KUKA KRL program: f1_Kuka_APT209T03S09.SRC

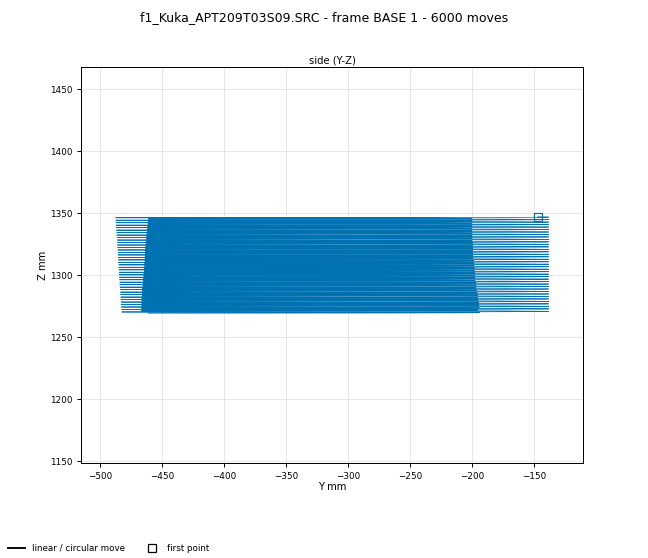
[picture p0: tool path of f1_Kuka_APT209T03S09.SRC in frame BASE 1, 6000 of 6001 moves have a stored position in this frame; points joined in program order, loops and branches not executed]
&ACCESS RVP
&REL 2
&PARAM TEMPLATE = C:\KRC\Roboter\Template\vorgabe
&PARAM EDITMASK = *
DEF f1_Kuka_APT209T03S09()


;FOLD INI;%{PE}%V3.2.0,%MKUKATPBASIS,%CINIT,%VCOMMON,%P
  ;FOLD BAS INI;%{E}%V3.2.0,%MKUKATPBASIS,%CINIT,%VINIT,%P
    GLOBAL INTERRUPT DECL 3 WHEN $STOPMESS==TRUE DO IR_STOPM ( )
    INTERRUPT ON 3
    BAS (#INITMOV,0 )
  ;ENDFOLD (BAS INI)
  ;FOLD USER INI;%{E}%V3.2.0,%MKUKATPUSER,%CINIT,%VINIT,%P
    ;Make your modifications here
  ;ENDFOLD (USER INI)
;ENDFOLD (INI)


;*** Make Null PTP Move
  PTP $pos_act

;*** Auto Load The Correct TOOL Data
  $tool=tool_data[3]

;*** Auto Load The Correct BASE Data
  $base=base_data[1]

  $ADVANCE = 5

;*** Restate Last Velocity
MMPM(30000.0)
SetRPM(6000)
LIN {X -0.021,Y -147.114,Z 1347.213,A 0.000,B 0.000,C 90.000,E1 218.382} C_DIS
LIN {X -0.029,Y -145.680,Z 1347.198,A 0.000,B 0.000,C 90.000,E1 215.644} C_DIS
LIN {X -0.031,Y -143.062,Z 1347.172,A 0.000,B 0.000,C 90.000,E1 211.052} C_DIS
LIN {X 0.026,Y -141.683,Z 1347.152,A 0.000,B 0.000,C 90.000,E1 207.334} C_DIS
LIN {X 0.005,Y -139.458,Z 1347.116,A 0.000,B 0.000,C 90.000,E1 200.844} C_DIS
LIN {X 0.056,Y -139.192,Z 1347.105,A 0.000,B 0.000,C 90.000,E1 198.960} C_DIS
LIN {X -0.057,Y -138.325,Z 1347.054,A 0.000,B 0.000,C 90.000,E1 189.670} C_DIS
LIN {X -0.053,Y -139.455,Z 1347.007,A 0.000,B 0.000,C 90.000,E1 181.260} C_DIS
LIN {X 0.027,Y -141.003,Z 1346.976,A 0.000,B 0.000,C 90.000,E1 175.641} C_DIS
LIN {X -0.023,Y -142.757,Z 1346.955,A 0.000,B 0.000,C 90.000,E1 171.951} C_DIS
LIN {X -0.068,Y -145.160,Z 1346.930,A 0.000,B 0.000,C 90.000,E1 167.353} C_DIS
LIN {X -0.076,Y -147.782,Z 1346.909,A 0.000,B 0.000,C 90.000,E1 163.685} C_DIS
LIN {X 0.003,Y -150.461,Z 1346.889,A 0.000,B 0.000,C 90.000,E1 160.007} C_DIS
LIN {X 0.079,Y -153.912,Z 1346.869,A 0.000,B 0.000,C 90.000,E1 156.357} C_DIS
LIN {X 0.003,Y -157.323,Z 1346.849,A 0.000,B 0.000,C 90.000,E1 152.794} C_DIS
LIN {X 0.087,Y -161.511,Z 1346.829,A 0.000,B 0.000,C 90.000,E1 149.203} C_DIS
LIN {X -0.036,Y -165.710,Z 1346.809,A 0.000,B 0.000,C 90.000,E1 145.722} C_DIS
LIN {X 0.089,Y -170.656,Z 1346.790,A 0.000,B 0.000,C 90.000,E1 142.190} C_DIS
LIN {X 0.002,Y -175.533,Z 1346.771,A 0.000,B 0.000,C 90.000,E1 138.771} C_DIS
LIN {X -0.004,Y -181.152,Z 1346.752,A 0.000,B 0.000,C 90.000,E1 135.364} C_DIS
LIN {X -0.007,Y -186.605,Z 1346.733,A 0.000,B 0.000,C 90.000,E1 132.000} C_DIS
LIN {X 0.063,Y -191.214,Z 1346.719,A 0.000,B 0.000,C 90.000,E1 129.483} C_DIS
LIN {X -0.013,Y -197.028,Z 1346.701,A 0.000,B 0.000,C 90.000,E1 126.217} C_DIS
LIN {X 0.060,Y -199.188,Z 1346.695,A 0.000,B 0.000,C 90.000,E1 125.105} C_DIS
LIN {X 0.058,Y -308.836,Z 1346.695,A 0.000,B 0.000,C 90.000,E1 125.105} C_DIS
LIN {X -0.131,Y -311.015,Z 1346.695,A 0.000,B 0.000,C 90.000,E1 125.105} C_DIS
LIN {X 0.079,Y -315.979,Z 1346.693,A 0.000,B 0.000,C 90.000,E1 124.818} C_DIS
LIN {X -0.152,Y -318.679,Z 1346.692,A 0.000,B 0.000,C 90.000,E1 124.612} C_DIS
LIN {X -0.061,Y -322.397,Z 1346.689,A 0.000,B 0.000,C 90.000,E1 124.072} C_DIS
LIN {X 0.196,Y -323.974,Z 1346.688,A 0.000,B 0.000,C 90.000,E1 123.706} C_DIS
LIN {X 0.124,Y -329.656,Z 1346.679,A 0.000,B 0.000,C 90.000,E1 122.133} C_DIS
LIN {X 0.058,Y -340.607,Z 1346.663,A 0.000,B 0.000,C 90.000,E1 119.333} C_DIS
LIN {X 0.113,Y -352.941,Z 1346.648,A 0.000,B 0.000,C 90.000,E1 116.565} C_DIS
LIN {X -0.104,Y -366.760,Z 1346.633,A 0.000,B 0.000,C 90.000,E1 113.898} C_DIS
LIN {X -0.018,Y -380.391,Z 1346.620,A 0.000,B 0.000,C 90.000,E1 111.535} C_DIS
LIN {X 0.139,Y -395.388,Z 1346.607,A 0.000,B 0.000,C 90.000,E1 109.214} C_DIS
LIN {X 0.038,Y -411.854,Z 1346.594,A 0.000,B 0.000,C 90.000,E1 106.985} C_DIS
LIN {X 0.222,Y -429.907,Z 1346.582,A 0.000,B 0.000,C 90.000,E1 104.773} C_DIS
LIN {X -0.080,Y -449.484,Z 1346.571,A 0.000,B 0.000,C 90.000,E1 102.703} C_DIS
LIN {X 0.151,Y -469.762,Z 1346.560,A 0.000,B 0.000,C 90.000,E1 100.725} C_DIS
LIN {X -0.162,Y -480.082,Z 1346.555,A 0.000,B 0.000,C 90.000,E1 99.849} C_DIS
LIN {X -0.063,Y -482.184,Z 1346.553,A 0.000,B 0.000,C 90.000,E1 99.613} C_DIS
LIN {X -0.184,Y -483.945,Z 1346.552,A 0.000,B 0.000,C 90.000,E1 99.378} C_DIS
LIN {X 0.095,Y -485.266,Z 1346.551,A 0.000,B 0.000,C 90.000,E1 99.095} C_DIS
LIN {X -0.127,Y -486.906,Z 1346.548,A 0.000,B 0.000,C 90.000,E1 98.624} C_DIS
LIN {X 0.065,Y -487.471,Z 1346.545,A 0.000,B 0.000,C 90.000,E1 98.106} C_DIS
LIN {X -0.214,Y -487.053,Z 1346.542,A 0.000,B 0.000,C 90.000,E1 97.644} C_DIS
LIN {X -0.007,Y -485.591,Z 1346.540,A 0.000,B 0.000,C 90.000,E1 97.125} C_DIS
LIN {X -0.116,Y -484.390,Z 1346.538,A 0.000,B 0.000,C 90.000,E1 96.891} C_DIS
LIN {X 0.079,Y -480.928,Z 1346.535,A 0.000,B 0.000,C 90.000,E1 96.372} C_DIS
LIN {X -0.128,Y -468.644,Z 1346.526,A 0.000,B 0.000,C 90.000,E1 94.645} C_DIS
LIN {X -0.194,Y -460.372,Z 1346.519,A 0.000,B 0.000,C 90.000,E1 93.383} C_DIS
LIN {X -0.018,Y -442.160,Z 1346.503,A 0.000,B 0.000,C 90.000,E1 90.516} C_DIS
LIN {X -0.118,Y -427.307,Z 1346.488,A 0.000,B 0.000,C 90.000,E1 87.879} C_DIS
LIN {X -0.104,Y -417.153,Z 1346.478,A 0.000,B 0.000,C 90.000,E1 85.988} C_DIS
LIN {X 0.161,Y -406.849,Z 1346.467,A 0.000,B 0.000,C 90.000,E1 84.033} C_DIS
LIN {X -0.175,Y -397.806,Z 1346.458,A 0.000,B 0.000,C 90.000,E1 82.413} C_DIS
LIN {X 0.118,Y -388.604,Z 1346.448,A 0.000,B 0.000,C 90.000,E1 80.679} C_DIS
LIN {X -0.083,Y -379.155,Z 1346.439,A 0.000,B 0.000,C 90.000,E1 78.993} C_DIS
LIN {X 0.068,Y -369.496,Z 1346.429,A 0.000,B 0.000,C 90.000,E1 77.229} C_DIS
LIN {X 0.006,Y -357.966,Z 1346.418,A 0.000,B 0.000,C 90.000,E1 75.172} C_DIS
LIN {X -0.113,Y -346.459,Z 1346.406,A 0.000,B 0.000,C 90.000,E1 73.087} C_DIS
LIN {X 0.053,Y -334.769,Z 1346.394,A 0.000,B 0.000,C 90.000,E1 70.913} C_DIS
LIN {X 0.078,Y -323.286,Z 1346.382,A 0.000,B 0.000,C 90.000,E1 68.720} C_DIS
LIN {X -0.120,Y -306.185,Z 1346.362,A 0.000,B 0.000,C 90.000,E1 65.229} C_DIS
LIN {X -0.076,Y -296.339,Z 1346.349,A 0.000,B 0.000,C 90.000,E1 62.922} C_DIS
LIN {X -0.095,Y -288.786,Z 1346.338,A 0.000,B 0.000,C 90.000,E1 60.923} C_DIS
LIN {X 0.023,Y -281.931,Z 1346.327,A 0.000,B 0.000,C 90.000,E1 58.869} C_DIS
LIN {X -0.138,Y -271.800,Z 1346.308,A 0.000,B 0.000,C 90.000,E1 55.468} C_DIS
LIN {X -0.041,Y -262.409,Z 1346.289,A 0.000,B 0.000,C 90.000,E1 51.949} C_DIS
LIN {X -0.118,Y -253.519,Z 1346.269,A 0.000,B 0.000,C 90.000,E1 48.405} C_DIS
LIN {X -0.011,Y -245.175,Z 1346.249,A 0.000,B 0.000,C 90.000,E1 44.757} C_DIS
LIN {X 0.013,Y -237.527,Z 1346.228,A 0.000,B 0.000,C 90.000,E1 41.067} C_DIS
LIN {X 0.054,Y -230.665,Z 1346.207,A 0.000,B 0.000,C 90.000,E1 37.317} C_DIS
LIN {X 0.153,Y -224.658,Z 1346.186,A 0.000,B 0.000,C 90.000,E1 33.499} C_DIS
LIN {X 0.131,Y -219.690,Z 1346.165,A 0.000,B 0.000,C 90.000,E1 29.667} C_DIS
LIN {X 0.066,Y -215.042,Z 1346.139,A 0.000,B 0.000,C 90.000,E1 25.027} C_DIS
LIN {X -0.033,Y -211.493,Z 1346.113,A 0.000,B 0.000,C 90.000,E1 20.355} C_DIS
LIN {X 0.064,Y -208.962,Z 1346.091,A 0.000,B 0.000,C 90.000,E1 16.386} C_DIS
LIN {X 0.106,Y -206.550,Z 1346.069,A 0.000,B 0.000,C 90.000,E1 12.411} C_DIS
LIN {X 0.007,Y -204.341,Z 1346.047,A 0.000,B 0.000,C 90.000,E1 8.454} C_DIS
LIN {X -0.064,Y -202.124,Z 1346.020,A 0.000,B 0.000,C 90.000,E1 3.669} C_DIS
LIN {X -0.057,Y -200.683,Z 1345.988,A 0.000,B 0.000,C 90.000,E1 357.936} C_DIS
LIN {X -0.077,Y -200.557,Z 1345.953,A 0.000,B 0.000,C 90.000,E1 351.489} C_DIS
LIN {X 0.019,Y -202.765,Z 1345.912,A 0.000,B 0.000,C 90.000,E1 344.212} C_DIS
LIN {X 0.067,Y -206.427,Z 1345.881,A 0.000,B 0.000,C 90.000,E1 338.592} C_DIS
LIN {X -0.106,Y -210.232,Z 1345.859,A 0.000,B 0.000,C 90.000,E1 334.665} C_DIS
LIN {X -0.083,Y -215.076,Z 1345.837,A 0.000,B 0.000,C 90.000,E1 330.717} C_DIS
LIN {X 0.041,Y -221.062,Z 1345.816,A 0.000,B 0.000,C 90.000,E1 326.786} C_DIS
LIN {X 0.102,Y -228.174,Z 1345.794,A 0.000,B 0.000,C 90.000,E1 322.924} C_DIS
LIN {X -0.060,Y -236.414,Z 1345.773,A 0.000,B 0.000,C 90.000,E1 319.175} C_DIS
LIN {X -0.018,Y -244.846,Z 1345.755,A 0.000,B 0.000,C 90.000,E1 315.810} C_DIS
LIN {X 0.115,Y -253.283,Z 1345.738,A 0.000,B 0.000,C 90.000,E1 312.852} C_DIS
LIN {X -0.047,Y -263.012,Z 1345.722,A 0.000,B 0.000,C 90.000,E1 310.011} C_DIS
LIN {X 0.023,Y -272.626,Z 1345.708,A 0.000,B 0.000,C 90.000,E1 307.523} C_DIS
LIN {X -0.011,Y -283.429,Z 1345.695,A 0.000,B 0.000,C 90.000,E1 305.105} C_DIS
LIN {X 0.139,Y -291.935,Z 1345.686,A 0.000,B 0.000,C 90.000,E1 303.372} C_DIS
LIN {X 0.030,Y -303.488,Z 1345.674,A 0.000,B 0.000,C 90.000,E1 301.386} C_DIS
LIN {X -0.014,Y -312.061,Z 1345.667,A 0.000,B 0.000,C 90.000,E1 300.079} C_DIS
LIN {X 0.060,Y -321.507,Z 1345.660,A 0.000,B 0.000,C 90.000,E1 298.771} C_DIS
LIN {X -0.126,Y -339.453,Z 1345.648,A 0.000,B 0.000,C 90.000,E1 296.616} C_DIS
LIN {X 0.065,Y -355.465,Z 1345.638,A 0.000,B 0.000,C 90.000,E1 294.771} C_DIS
LIN {X -0.108,Y -368.559,Z 1345.630,A 0.000,B 0.000,C 90.000,E1 293.334} C_DIS
LIN {X 0.060,Y -378.763,Z 1345.623,A 0.000,B 0.000,C 90.000,E1 292.153} C_DIS
LIN {X -0.141,Y -391.154,Z 1345.615,A 0.000,B 0.000,C 90.000,E1 290.737} C_DIS
LIN {X 0.096,Y -408.316,Z 1345.604,A 0.000,B 0.000,C 90.000,E1 288.725} C_DIS
LIN {X 0.076,Y -420.515,Z 1345.596,A 0.000,B 0.000,C 90.000,E1 287.347} C_DIS
LIN {X 0.078,Y -429.793,Z 1345.590,A 0.000,B 0.000,C 90.000,E1 286.260} C_DIS
LIN {X -0.126,Y -436.230,Z 1345.586,A 0.000,B 0.000,C 90.000,E1 285.481} C_DIS
LIN {X 0.040,Y -442.070,Z 1345.582,A 0.000,B 0.000,C 90.000,E1 284.662} C_DIS
LIN {X -0.060,Y -447.229,Z 1345.577,A 0.000,B 0.000,C 90.000,E1 283.883} C_DIS
LIN {X 0.216,Y -451.529,Z 1345.573,A 0.000,B 0.000,C 90.000,E1 283.063} C_DIS
LIN {X 0.091,Y -455.098,Z 1345.568,A 0.000,B 0.000,C 90.000,E1 282.299} C_DIS
LIN {X 0.175,Y -457.056,Z 1345.566,A 0.000,B 0.000,C 90.000,E1 281.771} C_DIS
LIN {X -0.185,Y -458.644,Z 1345.563,A 0.000,B 0.000,C 90.000,E1 281.299} C_DIS
LIN {X -0.174,Y -459.895,Z 1345.560,A 0.000,B 0.000,C 90.000,E1 280.782} C_DIS
LIN {X -0.064,Y -460.730,Z 1345.557,A 0.000,B 0.000,C 90.000,E1 280.254} C_DIS
LIN {X 0.049,Y -461.072,Z 1345.554,A 0.000,B 0.000,C 90.000,E1 279.726} C_DIS
LIN {X 0.090,Y -460.985,Z 1345.551,A 0.000,B 0.000,C 90.000,E1 279.208} C_DIS
LIN {X 0.136,Y -460.415,Z 1345.548,A 0.000,B 0.000,C 90.000,E1 278.690} C_DIS
LIN {X -0.204,Y -459.357,Z 1345.546,A 0.000,B 0.000,C 90.000,E1 278.219} C_DIS
LIN {X -0.161,Y -457.815,Z 1345.543,A 0.000,B 0.000,C 90.000,E1 277.701} C_DIS
LIN {X -0.121,Y -455.710,Z 1345.540,A 0.000,B 0.000,C 90.000,E1 277.182} C_DIS
LIN {X -0.089,Y -453.108,Z 1345.537,A 0.000,B 0.000,C 90.000,E1 276.663} C_DIS
LIN {X -0.077,Y -449.941,Z 1345.534,A 0.000,B 0.000,C 90.000,E1 276.144} C_DIS
LIN {X -0.081,Y -446.043,Z 1345.531,A 0.000,B 0.000,C 90.000,E1 275.625} C_DIS
LIN {X 0.149,Y -443.825,Z 1345.530,A 0.000,B 0.000,C 90.000,E1 275.334} C_DIS
LIN {X 0.101,Y -438.554,Z 1345.527,A 0.000,B 0.000,C 90.000,E1 274.821} C_DIS
LIN {X -0.109,Y -432.593,Z 1345.524,A 0.000,B 0.000,C 90.000,E1 274.359} C_DIS
LIN {X 0.100,Y -426.339,Z 1345.522,A 0.000,B 0.000,C 90.000,E1 273.898} C_DIS
LIN {X -0.180,Y -419.917,Z 1345.520,A 0.000,B 0.000,C 90.000,E1 273.555} C_DIS
LIN {X -0.126,Y -413.411,Z 1345.518,A 0.000,B 0.000,C 90.000,E1 273.212} C_DIS
LIN {X -0.185,Y -406.801,Z 1345.516,A 0.000,B 0.000,C 90.000,E1 272.922} C_DIS
LIN {X -0.038,Y -399.961,Z 1345.515,A 0.000,B 0.000,C 90.000,E1 272.636} C_DIS
LIN {X -0.062,Y -392.788,Z 1345.513,A 0.000,B 0.000,C 90.000,E1 272.407} C_DIS
LIN {X 0.153,Y -385.437,Z 1345.512,A 0.000,B 0.000,C 90.000,E1 272.178} C_DIS
LIN {X -0.160,Y -377.984,Z 1345.511,A 0.000,B 0.000,C 90.000,E1 272.064} C_DIS
LIN {X 0.109,Y -370.034,Z 1345.511,A 0.000,B 0.000,C 90.000,E1 271.892} C_DIS
LIN {X 0.185,Y -360.435,Z 1345.510,A 0.000,B 0.000,C 90.000,E1 271.776} C_DIS
LIN {X 0.022,Y -348.181,Z 1345.510,A 0.000,B 0.000,C 90.000,E1 271.718} C_DIS
LIN {X -0.034,Y -344.123,Z 1345.510,A 0.000,B 0.000,C 90.000,E1 271.718} C_DIS
LIN {X -0.048,Y -181.313,Z 1345.510,A 0.000,B 0.000,C 90.000,E1 271.718} C_DIS
LIN {X -0.004,Y -181.579,Z 1345.501,A 0.000,B 0.000,C 90.000,E1 270.172} C_DIS
LIN {X -0.045,Y -180.907,Z 1345.475,A 0.000,B 0.000,C 90.000,E1 265.469} C_DIS
LIN {X 0.011,Y -180.729,Z 1345.470,A 0.000,B 0.000,C 90.000,E1 264.609} C_DIS
LIN {X -0.066,Y -178.819,Z 1345.442,A 0.000,B 0.000,C 90.000,E1 259.567} C_DIS
LIN {X 0.015,Y -175.864,Z 1345.414,A 0.000,B 0.000,C 90.000,E1 254.448} C_DIS
LIN {X 0.064,Y -173.831,Z 1345.399,A 0.000,B 0.000,C 90.000,E1 251.873} C_DIS
LIN {X -0.001,Y -171.499,Z 1345.380,A 0.000,B 0.000,C 90.000,E1 248.465} C_DIS
LIN {X -0.014,Y -167.727,Z 1345.356,A 0.000,B 0.000,C 90.000,E1 244.152} C_DIS
LIN {X 0.002,Y -166.421,Z 1345.347,A 0.000,B 0.000,C 90.000,E1 242.410} C_DIS
LIN {X 0.000,Y -163.143,Z 1345.327,A 0.000,B 0.000,C 90.000,E1 238.918} C_DIS
LIN {X -0.034,Y -161.097,Z 1345.313,A 0.000,B 0.000,C 90.000,E1 236.294} C_DIS
LIN {X -0.051,Y -157.826,Z 1345.293,A 0.000,B 0.000,C 90.000,E1 232.763} C_DIS
LIN {X 0.013,Y -155.859,Z 1345.278,A 0.000,B 0.000,C 90.000,E1 230.070} C_DIS
LIN {X 0.069,Y -152.109,Z 1345.253,A 0.000,B 0.000,C 90.000,E1 225.567} C_DIS
LIN {X -0.024,Y -150.360,Z 1345.238,A 0.000,B 0.000,C 90.000,E1 222.894} C_DIS
LIN {X 0.015,Y -147.095,Z 1345.213,A 0.000,B 0.000,C 90.000,E1 218.338} C_DIS
LIN {X 0.010,Y -145.665,Z 1345.198,A 0.000,B 0.000,C 90.000,E1 215.598} C_DIS
LIN {X 0.012,Y -143.047,Z 1345.172,A 0.000,B 0.000,C 90.000,E1 211.003} C_DIS
LIN {X 0.013,Y -141.671,Z 1345.152,A 0.000,B 0.000,C 90.000,E1 207.308} C_DIS
LIN {X 0.057,Y -139.452,Z 1345.116,A 0.000,B 0.000,C 90.000,E1 200.791} C_DIS
LIN {X -0.021,Y -139.186,Z 1345.105,A 0.000,B 0.000,C 90.000,E1 198.960} C_DIS
LIN {X 0.001,Y -138.323,Z 1345.053,A 0.000,B 0.000,C 90.000,E1 189.613} C_DIS
LIN {X 0.009,Y -139.460,Z 1345.007,A 0.000,B 0.000,C 90.000,E1 181.203} C_DIS
LIN {X -0.051,Y -141.016,Z 1344.976,A 0.000,B 0.000,C 90.000,E1 175.641} C_DIS
LIN {X 0.039,Y -142.770,Z 1344.955,A 0.000,B 0.000,C 90.000,E1 171.894} C_DIS
LIN {X -0.006,Y -145.180,Z 1344.929,A 0.000,B 0.000,C 90.000,E1 167.297} C_DIS
LIN {X 0.028,Y -147.802,Z 1344.909,A 0.000,B 0.000,C 90.000,E1 163.614} C_DIS
LIN {X -0.077,Y -150.488,Z 1344.889,A 0.000,B 0.000,C 90.000,E1 160.007} C_DIS
LIN {X -0.005,Y -153.943,Z 1344.869,A 0.000,B 0.000,C 90.000,E1 156.357} C_DIS
LIN {X 0.059,Y -157.354,Z 1344.849,A 0.000,B 0.000,C 90.000,E1 152.743} C_DIS
LIN {X 0.002,Y -161.550,Z 1344.829,A 0.000,B 0.000,C 90.000,E1 149.203} C_DIS
LIN {X 0.014,Y -165.749,Z 1344.809,A 0.000,B 0.000,C 90.000,E1 145.674} C_DIS
LIN {X 0.001,Y -170.703,Z 1344.790,A 0.000,B 0.000,C 90.000,E1 142.190} C_DIS
LIN {X -0.087,Y -175.576,Z 1344.771,A 0.000,B 0.000,C 90.000,E1 138.771} C_DIS
LIN {X 0.032,Y -181.194,Z 1344.752,A 0.000,B 0.000,C 90.000,E1 135.324} C_DIS
LIN {X 0.025,Y -186.656,Z 1344.733,A 0.000,B 0.000,C 90.000,E1 131.962} C_DIS
LIN {X -0.030,Y -191.260,Z 1344.719,A 0.000,B 0.000,C 90.000,E1 129.483} C_DIS
LIN {X 0.050,Y -197.081,Z 1344.701,A 0.000,B 0.000,C 90.000,E1 126.171} C_DIS
LIN {X 0.064,Y -199.186,Z 1344.695,A 0.000,B 0.000,C 90.000,E1 125.105} C_DIS
LIN {X 0.051,Y -308.995,Z 1344.695,A 0.000,B 0.000,C 90.000,E1 125.105} C_DIS
LIN {X -0.017,Y -313.722,Z 1344.694,A 0.000,B 0.000,C 90.000,E1 124.978} C_DIS
LIN {X 0.094,Y -315.921,Z 1344.693,A 0.000,B 0.000,C 90.000,E1 124.818} C_DIS
LIN {X 0.138,Y -318.909,Z 1344.692,A 0.000,B 0.000,C 90.000,E1 124.532} C_DIS
LIN {X -0.072,Y -322.563,Z 1344.689,A 0.000,B 0.000,C 90.000,E1 124.040} C_DIS
LIN {X 0.004,Y -324.099,Z 1344.687,A 0.000,B 0.000,C 90.000,E1 123.706} C_DIS
LIN {X 0.044,Y -338.170,Z 1344.666,A 0.000,B 0.000,C 90.000,E1 119.922} C_DIS
LIN {X 0.185,Y -350.204,Z 1344.651,A 0.000,B 0.000,C 90.000,E1 117.129} C_DIS
LIN {X -0.111,Y -363.701,Z 1344.636,A 0.000,B 0.000,C 90.000,E1 114.463} C_DIS
LIN {X 0.039,Y -377.023,Z 1344.623,A 0.000,B 0.000,C 90.000,E1 112.078} C_DIS
LIN {X 0.104,Y -391.687,Z 1344.610,A 0.000,B 0.000,C 90.000,E1 109.758} C_DIS
LIN {X 0.033,Y -407.796,Z 1344.597,A 0.000,B 0.000,C 90.000,E1 107.511} C_DIS
LIN {X -0.008,Y -425.462,Z 1344.585,A 0.000,B 0.000,C 90.000,E1 105.315} C_DIS
LIN {X 0.025,Y -444.744,Z 1344.573,A 0.000,B 0.000,C 90.000,E1 103.175} C_DIS
LIN {X 0.025,Y -464.891,Z 1344.562,A 0.000,B 0.000,C 90.000,E1 101.186} C_DIS
LIN {X 0.106,Y -480.303,Z 1344.554,A 0.000,B 0.000,C 90.000,E1 99.792} C_DIS
LIN {X 0.208,Y -482.314,Z 1344.553,A 0.000,B 0.000,C 90.000,E1 99.557} C_DIS
LIN {X 0.089,Y -484.007,Z 1344.552,A 0.000,B 0.000,C 90.000,E1 99.321} C_DIS
LIN {X -0.108,Y -485.277,Z 1344.550,A 0.000,B 0.000,C 90.000,E1 99.095} C_DIS
LIN {X 0.151,Y -486.837,Z 1344.548,A 0.000,B 0.000,C 90.000,E1 98.568} C_DIS
LIN {X -0.140,Y -487.334,Z 1344.545,A 0.000,B 0.000,C 90.000,E1 98.106} C_DIS
LIN {X 0.064,Y -486.850,Z 1344.542,A 0.000,B 0.000,C 90.000,E1 97.587} C_DIS
LIN {X -0.212,Y -485.310,Z 1344.539,A 0.000,B 0.000,C 90.000,E1 97.125} C_DIS
LIN {X 0.160,Y -484.062,Z 1344.538,A 0.000,B 0.000,C 90.000,E1 96.834} C_DIS
LIN {X -0.126,Y -480.536,Z 1344.535,A 0.000,B 0.000,C 90.000,E1 96.372} C_DIS
LIN {X 0.133,Y -468.268,Z 1344.526,A 0.000,B 0.000,C 90.000,E1 94.588} C_DIS
LIN {X -0.131,Y -458.280,Z 1344.517,A 0.000,B 0.000,C 90.000,E1 93.094} C_DIS
LIN {X 0.211,Y -441.778,Z 1344.503,A 0.000,B 0.000,C 90.000,E1 90.458} C_DIS
LIN {X 0.093,Y -426.949,Z 1344.488,A 0.000,B 0.000,C 90.000,E1 87.822} C_DIS
LIN {X 0.123,Y -416.806,Z 1344.477,A 0.000,B 0.000,C 90.000,E1 85.927} C_DIS
LIN {X -0.058,Y -406.499,Z 1344.467,A 0.000,B 0.000,C 90.000,E1 84.033} C_DIS
LIN {X 0.074,Y -395.956,Z 1344.456,A 0.000,B 0.000,C 90.000,E1 82.064} C_DIS
LIN {X -0.054,Y -386.708,Z 1344.447,A 0.000,B 0.000,C 90.000,E1 80.387} C_DIS
LIN {X 0.160,Y -377.221,Z 1344.437,A 0.000,B 0.000,C 90.000,E1 78.634} C_DIS
LIN {X -0.162,Y -367.490,Z 1344.427,A 0.000,B 0.000,C 90.000,E1 76.937} C_DIS
LIN {X 0.126,Y -354.341,Z 1344.414,A 0.000,B 0.000,C 90.000,E1 74.519} C_DIS
LIN {X 0.011,Y -344.435,Z 1344.404,A 0.000,B 0.000,C 90.000,E1 72.725} C_DIS
LIN {X 0.116,Y -331.122,Z 1344.390,A 0.000,B 0.000,C 90.000,E1 70.242} C_DIS
LIN {X 0.068,Y -316.555,Z 1344.375,A 0.000,B 0.000,C 90.000,E1 67.411} C_DIS
LIN {X -0.104,Y -301.544,Z 1344.357,A 0.000,B 0.000,C 90.000,E1 64.204} C_DIS
LIN {X 0.097,Y -292.173,Z 1344.344,A 0.000,B 0.000,C 90.000,E1 61.847} C_DIS
LIN {X 0.074,Y -282.796,Z 1344.329,A 0.000,B 0.000,C 90.000,E1 59.154} C_DIS
LIN {X 0.021,Y -271.612,Z 1344.308,A 0.000,B 0.000,C 90.000,E1 55.388} C_DIS
LIN {X -0.052,Y -262.256,Z 1344.288,A 0.000,B 0.000,C 90.000,E1 51.904} C_DIS
LIN {X 0.026,Y -253.407,Z 1344.269,A 0.000,B 0.000,C 90.000,E1 48.324} C_DIS
LIN {X 0.124,Y -245.100,Z 1344.248,A 0.000,B 0.000,C 90.000,E1 44.676} C_DIS
LIN {X -0.014,Y -237.470,Z 1344.228,A 0.000,B 0.000,C 90.000,E1 41.024} C_DIS
LIN {X -0.007,Y -230.618,Z 1344.207,A 0.000,B 0.000,C 90.000,E1 37.282} C_DIS
LIN {X -0.044,Y -224.624,Z 1344.186,A 0.000,B 0.000,C 90.000,E1 33.499} C_DIS
LIN {X -0.064,Y -219.698,Z 1344.165,A 0.000,B 0.000,C 90.000,E1 29.667} C_DIS
LIN {X -0.123,Y -215.063,Z 1344.139,A 0.000,B 0.000,C 90.000,E1 25.027} C_DIS
LIN {X -0.065,Y -212.048,Z 1344.117,A 0.000,B 0.000,C 90.000,E1 21.099} C_DIS
LIN {X -0.020,Y -209.415,Z 1344.095,A 0.000,B 0.000,C 90.000,E1 17.149} C_DIS
LIN {X -0.112,Y -207.446,Z 1344.078,A 0.000,B 0.000,C 90.000,E1 14.008} C_DIS
LIN {X -0.060,Y -205.083,Z 1344.056,A 0.000,B 0.000,C 90.000,E1 10.018} C_DIS
LIN {X -0.068,Y -203.049,Z 1344.033,A 0.000,B 0.000,C 90.000,E1 6.024} C_DIS
LIN {X -0.037,Y -200.922,Z 1343.997,A 0.000,B 0.000,C 90.000,E1 359.542} C_DIS
LIN {X -0.102,Y -200.420,Z 1343.962,A 0.000,B 0.000,C 90.000,E1 353.109} C_DIS
LIN {X 0.002,Y -202.110,Z 1343.921,A 0.000,B 0.000,C 90.000,E1 345.825} C_DIS
LIN {X 0.074,Y -205.294,Z 1343.890,A 0.000,B 0.000,C 90.000,E1 340.188} C_DIS
LIN {X 0.076,Y -209.518,Z 1343.864,A 0.000,B 0.000,C 90.000,E1 335.409} C_DIS
LIN {X -0.112,Y -214.168,Z 1343.842,A 0.000,B 0.000,C 90.000,E1 331.513} C_DIS
LIN {X -0.018,Y -219.925,Z 1343.820,A 0.000,B 0.000,C 90.000,E1 327.582} C_DIS
LIN {X 0.067,Y -226.801,Z 1343.798,A 0.000,B 0.000,C 90.000,E1 323.703} C_DIS
LIN {X 0.047,Y -234.832,Z 1343.777,A 0.000,B 0.000,C 90.000,E1 319.908} C_DIS
LIN {X 0.085,Y -242.036,Z 1343.761,A 0.000,B 0.000,C 90.000,E1 316.905} C_DIS
LIN {X -0.040,Y -251.183,Z 1343.742,A 0.000,B 0.000,C 90.000,E1 313.623} C_DIS
LIN {X 0.065,Y -259.317,Z 1343.728,A 0.000,B 0.000,C 90.000,E1 311.067} C_DIS
LIN {X 0.016,Y -268.456,Z 1343.714,A 0.000,B 0.000,C 90.000,E1 308.588} C_DIS
LIN {X 0.042,Y -278.751,Z 1343.701,A 0.000,B 0.000,C 90.000,E1 306.137} C_DIS
LIN {X 0.079,Y -288.548,Z 1343.689,A 0.000,B 0.000,C 90.000,E1 304.072} C_DIS
LIN {X -0.085,Y -295.771,Z 1343.682,A 0.000,B 0.000,C 90.000,E1 302.752} C_DIS
LIN {X 0.108,Y -305.644,Z 1343.673,A 0.000,B 0.000,C 90.000,E1 301.052} C_DIS
LIN {X 0.096,Y -314.419,Z 1343.665,A 0.000,B 0.000,C 90.000,E1 299.745} C_DIS
LIN {X -0.003,Y -326.562,Z 1343.656,A 0.000,B 0.000,C 90.000,E1 298.153} C_DIS
LIN {X -0.141,Y -347.440,Z 1343.643,A 0.000,B 0.000,C 90.000,E1 295.720} C_DIS
LIN {X 0.128,Y -360.517,Z 1343.635,A 0.000,B 0.000,C 90.000,E1 294.207} C_DIS
LIN {X -0.016,Y -373.499,Z 1343.626,A 0.000,B 0.000,C 90.000,E1 292.770} C_DIS
LIN {X 0.098,Y -383.627,Z 1343.620,A 0.000,B 0.000,C 90.000,E1 291.589} C_DIS
LIN {X 0.007,Y -395.839,Z 1343.612,A 0.000,B 0.000,C 90.000,E1 290.174} C_DIS
LIN {X -0.179,Y -413.074,Z 1343.601,A 0.000,B 0.000,C 90.000,E1 288.236} C_DIS
LIN {X -0.138,Y -425.064,Z 1343.594,A 0.000,B 0.000,C 90.000,E1 286.858} C_DIS
LIN {X -0.211,Y -434.007,Z 1343.588,A 0.000,B 0.000,C 90.000,E1 285.788} C_DIS
LIN {X 0.043,Y -440.048,Z 1343.583,A 0.000,B 0.000,C 90.000,E1 284.954} C_DIS
LIN {X -0.071,Y -445.482,Z 1343.579,A 0.000,B 0.000,C 90.000,E1 284.175} C_DIS
LIN {X 0.182,Y -450.148,Z 1343.574,A 0.000,B 0.000,C 90.000,E1 283.355} C_DIS
LIN {X 0.048,Y -453.953,Z 1343.570,A 0.000,B 0.000,C 90.000,E1 282.591} C_DIS
LIN {X -0.140,Y -455.105,Z 1343.568,A 0.000,B 0.000,C 90.000,E1 282.355} C_DIS
LIN {X -0.058,Y -457.070,Z 1343.566,A 0.000,B 0.000,C 90.000,E1 281.827} C_DIS
LIN {X 0.030,Y -458.722,Z 1343.563,A 0.000,B 0.000,C 90.000,E1 281.299} C_DIS
LIN {X 0.043,Y -460.009,Z 1343.560,A 0.000,B 0.000,C 90.000,E1 280.782} C_DIS
LIN {X 0.152,Y -460.852,Z 1343.557,A 0.000,B 0.000,C 90.000,E1 280.254} C_DIS
LIN {X -0.188,Y -461.277,Z 1343.554,A 0.000,B 0.000,C 90.000,E1 279.782} C_DIS
LIN {X -0.147,Y -461.237,Z 1343.551,A 0.000,B 0.000,C 90.000,E1 279.265} C_DIS
LIN {X -0.100,Y -460.758,Z 1343.548,A 0.000,B 0.000,C 90.000,E1 278.746} C_DIS
LIN {X 0.016,Y -459.730,Z 1343.546,A 0.000,B 0.000,C 90.000,E1 278.219} C_DIS
LIN {X 0.061,Y -458.252,Z 1343.543,A 0.000,B 0.000,C 90.000,E1 277.701} C_DIS
LIN {X 0.102,Y -456.210,Z 1343.540,A 0.000,B 0.000,C 90.000,E1 277.182} C_DIS
LIN {X 0.135,Y -453.689,Z 1343.537,A 0.000,B 0.000,C 90.000,E1 276.663} C_DIS
LIN {X 0.149,Y -450.564,Z 1343.534,A 0.000,B 0.000,C 90.000,E1 276.144} C_DIS
LIN {X 0.146,Y -446.777,Z 1343.531,A 0.000,B 0.000,C 90.000,E1 275.625} C_DIS
LIN {X -0.066,Y -444.598,Z 1343.530,A 0.000,B 0.000,C 90.000,E1 275.391} C_DIS
LIN {X -0.129,Y -439.434,Z 1343.527,A 0.000,B 0.000,C 90.000,E1 274.878} C_DIS
LIN {X 0.046,Y -433.568,Z 1343.524,A 0.000,B 0.000,C 90.000,E1 274.359} C_DIS
LIN {X 0.194,Y -427.378,Z 1343.522,A 0.000,B 0.000,C 90.000,E1 273.898} C_DIS
LIN {X -0.151,Y -420.932,Z 1343.520,A 0.000,B 0.000,C 90.000,E1 273.555} C_DIS
LIN {X -0.148,Y -414.384,Z 1343.518,A 0.000,B 0.000,C 90.000,E1 273.212} C_DIS
LIN {X 0.173,Y -407.809,Z 1343.516,A 0.000,B 0.000,C 90.000,E1 272.865} C_DIS
LIN {X -0.113,Y -401.003,Z 1343.515,A 0.000,B 0.000,C 90.000,E1 272.636} C_DIS
LIN {X -0.144,Y -393.880,Z 1343.513,A 0.000,B 0.000,C 90.000,E1 272.407} C_DIS
LIN {X 0.069,Y -386.676,Z 1343.512,A 0.000,B 0.000,C 90.000,E1 272.178} C_DIS
LIN {X 0.007,Y -375.090,Z 1343.511,A 0.000,B 0.000,C 90.000,E1 271.949} C_DIS
LIN {X -0.039,Y -366.188,Z 1343.510,A 0.000,B 0.000,C 90.000,E1 271.835} C_DIS
LIN {X -0.010,Y -352.971,Z 1343.510,A 0.000,B 0.000,C 90.000,E1 271.718} C_DIS
LIN {X 0.164,Y -345.765,Z 1343.509,A 0.000,B 0.000,C 90.000,E1 271.661} C_DIS
LIN {X 0.056,Y -181.318,Z 1343.509,A 0.000,B 0.000,C 90.000,E1 271.661} C_DIS
LIN {X -0.082,Y -181.577,Z 1343.501,A 0.000,B 0.000,C 90.000,E1 270.172} C_DIS
LIN {X 0.057,Y -180.906,Z 1343.475,A 0.000,B 0.000,C 90.000,E1 265.412} C_DIS
LIN {X -0.066,Y -180.719,Z 1343.470,A 0.000,B 0.000,C 90.000,E1 264.609} C_DIS
LIN {X 0.032,Y -178.806,Z 1343.442,A 0.000,B 0.000,C 90.000,E1 259.511} C_DIS
LIN {X -0.061,Y -175.851,Z 1343.413,A 0.000,B 0.000,C 90.000,E1 254.448} C_DIS
LIN {X -0.079,Y -173.177,Z 1343.395,A 0.000,B 0.000,C 90.000,E1 251.040} C_DIS
LIN {X -0.076,Y -171.478,Z 1343.380,A 0.000,B 0.000,C 90.000,E1 248.465} C_DIS
LIN {X -0.089,Y -167.708,Z 1343.356,A 0.000,B 0.000,C 90.000,E1 244.152} C_DIS
LIN {X 0.076,Y -166.396,Z 1343.347,A 0.000,B 0.000,C 90.000,E1 242.359} C_DIS
LIN {X 0.067,Y -163.122,Z 1343.327,A 0.000,B 0.000,C 90.000,E1 238.869} C_DIS
LIN {X -0.107,Y -161.072,Z 1343.313,A 0.000,B 0.000,C 90.000,E1 236.294} C_DIS
LIN {X 0.004,Y -157.804,Z 1343.293,A 0.000,B 0.000,C 90.000,E1 232.718} C_DIS
LIN {X -0.058,Y -155.840,Z 1343.278,A 0.000,B 0.000,C 90.000,E1 230.070} C_DIS
LIN {X -0.001,Y -152.091,Z 1343.253,A 0.000,B 0.000,C 90.000,E1 225.567} C_DIS
LIN {X 0.017,Y -150.340,Z 1343.238,A 0.000,B 0.000,C 90.000,E1 222.852} C_DIS
LIN {X 0.038,Y -147.080,Z 1343.213,A 0.000,B 0.000,C 90.000,E1 218.302} C_DIS
LIN {X -0.058,Y -145.653,Z 1343.198,A 0.000,B 0.000,C 90.000,E1 215.598} C_DIS
LIN {X -0.054,Y -143.035,Z 1343.172,A 0.000,B 0.000,C 90.000,E1 211.003} C_DIS
LIN {X 0.073,Y -141.660,Z 1343.152,A 0.000,B 0.000,C 90.000,E1 207.257} C_DIS
LIN {X -0.008,Y -139.447,Z 1343.115,A 0.000,B 0.000,C 90.000,E1 200.791} C_DIS
LIN {X 0.044,Y -139.181,Z 1343.105,A 0.000,B 0.000,C 90.000,E1 198.906} C_DIS
LIN {X -0.064,Y -138.321,Z 1343.053,A 0.000,B 0.000,C 90.000,E1 189.613} C_DIS
LIN {X -0.057,Y -139.465,Z 1343.007,A 0.000,B 0.000,C 90.000,E1 181.203} C_DIS
LIN {X 0.022,Y -141.027,Z 1342.975,A 0.000,B 0.000,C 90.000,E1 175.584} C_DIS
LIN {X -0.022,Y -142.393,Z 1342.960,A 0.000,B 0.000,C 90.000,E1 172.818} C_DIS
LIN {X 0.040,Y -144.624,Z 1342.934,A 0.000,B 0.000,C 90.000,E1 168.173} C_DIS
LIN {X -0.041,Y -147.819,Z 1342.909,A 0.000,B 0.000,C 90.000,E1 163.614} C_DIS
LIN {X 0.046,Y -150.510,Z 1342.889,A 0.000,B 0.000,C 90.000,E1 159.934} C_DIS
LIN {X -0.075,Y -153.969,Z 1342.869,A 0.000,B 0.000,C 90.000,E1 156.357} C_DIS
LIN {X -0.012,Y -157.382,Z 1342.849,A 0.000,B 0.000,C 90.000,E1 152.743} C_DIS
LIN {X -0.071,Y -161.584,Z 1342.829,A 0.000,B 0.000,C 90.000,E1 149.203} C_DIS
LIN {X -0.060,Y -165.781,Z 1342.809,A 0.000,B 0.000,C 90.000,E1 145.674} C_DIS
LIN {X -0.074,Y -170.743,Z 1342.790,A 0.000,B 0.000,C 90.000,E1 142.190} C_DIS
LIN {X 0.084,Y -175.615,Z 1342.771,A 0.000,B 0.000,C 90.000,E1 138.690} C_DIS
LIN {X -0.046,Y -181.231,Z 1342.752,A 0.000,B 0.000,C 90.000,E1 135.324} C_DIS
LIN {X 0.085,Y -186.699,Z 1342.733,A 0.000,B 0.000,C 90.000,E1 131.919} C_DIS
LIN {X 0.036,Y -191.299,Z 1342.719,A 0.000,B 0.000,C 90.000,E1 129.439} C_DIS
LIN {X -0.032,Y -197.128,Z 1342.701,A 0.000,B 0.000,C 90.000,E1 126.171} C_DIS
LIN {X 0.075,Y -199.179,Z 1342.695,A 0.000,B 0.000,C 90.000,E1 125.105} C_DIS
LIN {X 0.068,Y -308.381,Z 1342.695,A 0.000,B 0.000,C 90.000,E1 125.105} C_DIS
LIN {X -0.076,Y -310.577,Z 1342.695,A 0.000,B 0.000,C 90.000,E1 125.105} C_DIS
LIN {X -0.036,Y -316.211,Z 1342.693,A 0.000,B 0.000,C 90.000,E1 124.818} C_DIS
LIN {X 0.006,Y -319.097,Z 1342.692,A 0.000,B 0.000,C 90.000,E1 124.532} C_DIS
LIN {X -0.021,Y -322.748,Z 1342.689,A 0.000,B 0.000,C 90.000,E1 123.992} C_DIS
LIN {X 0.058,Y -324.237,Z 1342.687,A 0.000,B 0.000,C 90.000,E1 123.658} C_DIS
LIN {X -0.021,Y -337.048,Z 1342.668,A 0.000,B 0.000,C 90.000,E1 120.207} C_DIS
LIN {X -0.050,Y -348.943,Z 1342.652,A 0.000,B 0.000,C 90.000,E1 117.436} C_DIS
LIN {X -0.073,Y -362.294,Z 1342.637,A 0.000,B 0.000,C 90.000,E1 114.719} C_DIS
LIN {X 0.046,Y -375.473,Z 1342.624,A 0.000,B 0.000,C 90.000,E1 112.333} C_DIS
LIN {X 0.211,Y -389.986,Z 1342.611,A 0.000,B 0.000,C 90.000,E1 109.993} C_DIS
LIN {X -0.027,Y -405.931,Z 1342.599,A 0.000,B 0.000,C 90.000,E1 107.764} C_DIS
LIN {X 0.007,Y -423.421,Z 1342.586,A 0.000,B 0.000,C 90.000,E1 105.552} C_DIS
LIN {X -0.043,Y -442.554,Z 1342.574,A 0.000,B 0.000,C 90.000,E1 103.411} C_DIS
LIN {X -0.195,Y -462.638,Z 1342.563,A 0.000,B 0.000,C 90.000,E1 101.422} C_DIS
LIN {X -0.125,Y -480.536,Z 1342.554,A 0.000,B 0.000,C 90.000,E1 99.792} C_DIS
LIN {X -0.022,Y -482.454,Z 1342.553,A 0.000,B 0.000,C 90.000,E1 99.557} C_DIS
LIN {X -0.140,Y -484.077,Z 1342.552,A 0.000,B 0.000,C 90.000,E1 99.321} C_DIS
LIN {X 0.218,Y -485.292,Z 1342.550,A 0.000,B 0.000,C 90.000,E1 99.029} C_DIS
LIN {X -0.080,Y -486.770,Z 1342.547,A 0.000,B 0.000,C 90.000,E1 98.568} C_DIS
LIN {X 0.114,Y -487.195,Z 1342.545,A 0.000,B 0.000,C 90.000,E1 98.049} C_DIS
LIN {X -0.166,Y -486.641,Z 1342.542,A 0.000,B 0.000,C 90.000,E1 97.587} C_DIS
LIN {X 0.040,Y -485.018,Z 1342.539,A 0.000,B 0.000,C 90.000,E1 97.068} C_DIS
LIN {X -0.070,Y -483.716,Z 1342.538,A 0.000,B 0.000,C 90.000,E1 96.834} C_DIS
LIN {X -0.099,Y -467.860,Z 1342.525,A 0.000,B 0.000,C 90.000,E1 94.588} C_DIS
LIN {X 0.092,Y -457.866,Z 1342.517,A 0.000,B 0.000,C 90.000,E1 93.037} C_DIS
LIN {X -0.026,Y -441.386,Z 1342.503,A 0.000,B 0.000,C 90.000,E1 90.458} C_DIS
LIN {X -0.147,Y -426.569,Z 1342.488,A 0.000,B 0.000,C 90.000,E1 87.822} C_DIS
LIN {X -0.119,Y -416.438,Z 1342.477,A 0.000,B 0.000,C 90.000,E1 85.927} C_DIS
LIN {X 0.037,Y -407.622,Z 1342.468,A 0.000,B 0.000,C 90.000,E1 84.261} C_DIS
LIN {X 0.147,Y -397.118,Z 1342.457,A 0.000,B 0.000,C 90.000,E1 82.299} C_DIS
LIN {X 0.034,Y -387.881,Z 1342.448,A 0.000,B 0.000,C 90.000,E1 80.622} C_DIS
LIN {X -0.108,Y -378.437,Z 1342.438,A 0.000,B 0.000,C 90.000,E1 78.926} C_DIS
LIN {X -0.041,Y -368.748,Z 1342.429,A 0.000,B 0.000,C 90.000,E1 77.173} C_DIS
LIN {X -0.027,Y -357.222,Z 1342.417,A 0.000,B 0.000,C 90.000,E1 75.102} C_DIS
LIN {X -0.179,Y -347.369,Z 1342.407,A 0.000,B 0.000,C 90.000,E1 73.323} C_DIS
LIN {X 0.017,Y -337.352,Z 1342.397,A 0.000,B 0.000,C 90.000,E1 71.456} C_DIS
LIN {X 0.064,Y -324.200,Z 1342.383,A 0.000,B 0.000,C 90.000,E1 68.954} C_DIS
LIN {X 0.064,Y -307.055,Z 1342.364,A 0.000,B 0.000,C 90.000,E1 65.433} C_DIS
LIN {X 0.108,Y -297.120,Z 1342.351,A 0.000,B 0.000,C 90.000,E1 63.127} C_DIS
LIN {X 0.097,Y -289.452,Z 1342.340,A 0.000,B 0.000,C 90.000,E1 61.129} C_DIS
LIN {X -0.053,Y -281.482,Z 1342.327,A 0.000,B 0.000,C 90.000,E1 58.791} C_DIS
LIN {X 0.011,Y -271.410,Z 1342.307,A 0.000,B 0.000,C 90.000,E1 55.341} C_DIS
LIN {X 0.085,Y -262.092,Z 1342.288,A 0.000,B 0.000,C 90.000,E1 51.823} C_DIS
LIN {X 0.155,Y -253.294,Z 1342.268,A 0.000,B 0.000,C 90.000,E1 48.243} C_DIS
LIN {X -0.099,Y -245.025,Z 1342.248,A 0.000,B 0.000,C 90.000,E1 44.676} C_DIS
LIN {X -0.077,Y -237.403,Z 1342.228,A 0.000,B 0.000,C 90.000,E1 40.987} C_DIS
LIN {X -0.039,Y -230.560,Z 1342.207,A 0.000,B 0.000,C 90.000,E1 37.237} C_DIS
LIN {X 0.057,Y -224.585,Z 1342.186,A 0.000,B 0.000,C 90.000,E1 33.420} C_DIS
LIN {X 0.029,Y -219.675,Z 1342.164,A 0.000,B 0.000,C 90.000,E1 29.589} C_DIS
LIN {X -0.040,Y -215.071,Z 1342.139,A 0.000,B 0.000,C 90.000,E1 24.951} C_DIS
LIN {X -0.021,Y -211.487,Z 1342.112,A 0.000,B 0.000,C 90.000,E1 20.248} C_DIS
LIN {X -0.058,Y -208.869,Z 1342.091,A 0.000,B 0.000,C 90.000,E1 16.315} C_DIS
LIN {X 0.038,Y -206.890,Z 1342.073,A 0.000,B 0.000,C 90.000,E1 13.119} C_DIS
LIN {X -0.012,Y -204.536,Z 1342.051,A 0.000,B 0.000,C 90.000,E1 9.151} C_DIS
LIN {X -0.057,Y -202.589,Z 1342.029,A 0.000,B 0.000,C 90.000,E1 5.163} C_DIS
LIN {X -0.050,Y -200.696,Z 1341.993,A 0.000,B 0.000,C 90.000,E1 358.740} C_DIS
LIN {X -0.093,Y -200.476,Z 1341.957,A 0.000,B 0.000,C 90.000,E1 352.299} C_DIS
LIN {X -0.091,Y -202.509,Z 1341.917,A 0.000,B 0.000,C 90.000,E1 345.046} C_DIS
LIN {X 0.070,Y -205.988,Z 1341.886,A 0.000,B 0.000,C 90.000,E1 339.390} C_DIS
LIN {X 0.080,Y -209.635,Z 1341.864,A 0.000,B 0.000,C 90.000,E1 335.409} C_DIS
LIN {X -0.105,Y -214.307,Z 1341.842,A 0.000,B 0.000,C 90.000,E1 331.513} C_DIS
LIN {X -0.006,Y -220.073,Z 1341.820,A 0.000,B 0.000,C 90.000,E1 327.582} C_DIS
LIN {X 0.083,Y -226.939,Z 1341.798,A 0.000,B 0.000,C 90.000,E1 323.703} C_DIS
LIN {X 0.069,Y -234.972,Z 1341.777,A 0.000,B 0.000,C 90.000,E1 319.908} C_DIS
LIN {X -0.054,Y -242.156,Z 1341.761,A 0.000,B 0.000,C 90.000,E1 316.944} C_DIS
LIN {X -0.009,Y -251.296,Z 1341.742,A 0.000,B 0.000,C 90.000,E1 313.623} C_DIS
LIN {X 0.099,Y -259.426,Z 1341.728,A 0.000,B 0.000,C 90.000,E1 311.067} C_DIS
LIN {X 0.055,Y -268.551,Z 1341.714,A 0.000,B 0.000,C 90.000,E1 308.588} C_DIS
LIN {X -0.080,Y -278.844,Z 1341.701,A 0.000,B 0.000,C 90.000,E1 306.171} C_DIS
LIN {X -0.115,Y -288.659,Z 1341.689,A 0.000,B 0.000,C 90.000,E1 304.119} C_DIS
LIN {X -0.040,Y -297.798,Z 1341.680,A 0.000,B 0.000,C 90.000,E1 302.418} C_DIS
LIN {X 0.025,Y -307.890,Z 1341.671,A 0.000,B 0.000,C 90.000,E1 300.747} C_DIS
LIN {X -0.074,Y -316.856,Z 1341.664,A 0.000,B 0.000,C 90.000,E1 299.461} C_DIS
LIN {X 0.076,Y -329.073,Z 1341.655,A 0.000,B 0.000,C 90.000,E1 297.847} C_DIS
LIN {X -0.008,Y -347.363,Z 1341.643,A 0.000,B 0.000,C 90.000,E1 295.720} C_DIS
LIN {X -0.083,Y -360.435,Z 1341.635,A 0.000,B 0.000,C 90.000,E1 294.259} C_DIS
LIN {X 0.082,Y -373.418,Z 1341.627,A 0.000,B 0.000,C 90.000,E1 292.770} C_DIS
LIN {X 0.181,Y -383.579,Z 1341.620,A 0.000,B 0.000,C 90.000,E1 291.589} C_DIS
LIN {X 0.051,Y -395.817,Z 1341.612,A 0.000,B 0.000,C 90.000,E1 290.174} C_DIS
LIN {X -0.133,Y -413.055,Z 1341.601,A 0.000,B 0.000,C 90.000,E1 288.236} C_DIS
LIN {X -0.090,Y -425.055,Z 1341.594,A 0.000,B 0.000,C 90.000,E1 286.858} C_DIS
LIN {X -0.162,Y -434.012,Z 1341.588,A 0.000,B 0.000,C 90.000,E1 285.788} C_DIS
LIN {X 0.092,Y -440.074,Z 1341.583,A 0.000,B 0.000,C 90.000,E1 284.954} C_DIS
LIN {X -0.020,Y -445.511,Z 1341.579,A 0.000,B 0.000,C 90.000,E1 284.175} C_DIS
LIN {X 0.233,Y -450.189,Z 1341.574,A 0.000,B 0.000,C 90.000,E1 283.355} C_DIS
LIN {X -0.155,Y -452.858,Z 1341.571,A 0.000,B 0.000,C 90.000,E1 282.883} C_DIS
LIN {X -0.088,Y -455.184,Z 1341.569,A 0.000,B 0.000,C 90.000,E1 282.355} C_DIS
LIN {X -0.006,Y -457.157,Z 1341.566,A 0.000,B 0.000,C 90.000,E1 281.827} C_DIS
LIN {X 0.083,Y -458.821,Z 1341.563,A 0.000,B 0.000,C 90.000,E1 281.299} C_DIS
LIN {X 0.096,Y -460.114,Z 1341.560,A 0.000,B 0.000,C 90.000,E1 280.782} C_DIS
LIN {X 0.206,Y -461.013,Z 1341.557,A 0.000,B 0.000,C 90.000,E1 280.254} C_DIS
LIN {X -0.133,Y -461.459,Z 1341.554,A 0.000,B 0.000,C 90.000,E1 279.782} C_DIS
LIN {X -0.091,Y -461.499,Z 1341.551,A 0.000,B 0.000,C 90.000,E1 279.265} C_DIS
LIN {X -0.043,Y -461.012,Z 1341.549,A 0.000,B 0.000,C 90.000,E1 278.746} C_DIS
LIN {X 0.074,Y -460.055,Z 1341.546,A 0.000,B 0.000,C 90.000,E1 278.219} C_DIS
LIN {X 0.121,Y -458.600,Z 1341.543,A 0.000,B 0.000,C 90.000,E1 277.701} C_DIS
LIN {X 0.163,Y -456.680,Z 1341.540,A 0.000,B 0.000,C 90.000,E1 277.182} C_DIS
LIN {X 0.198,Y -454.132,Z 1341.537,A 0.000,B 0.000,C 90.000,E1 276.663} C_DIS
LIN {X 0.214,Y -451.045,Z 1341.534,A 0.000,B 0.000,C 90.000,E1 276.144} C_DIS
LIN {X 0.213,Y -447.332,Z 1341.531,A 0.000,B 0.000,C 90.000,E1 275.625} C_DIS
LIN {X 0.193,Y -442.820,Z 1341.529,A 0.000,B 0.000,C 90.000,E1 275.106} C_DIS
LIN {X 0.147,Y -437.239,Z 1341.526,A 0.000,B 0.000,C 90.000,E1 274.588} C_DIS
LIN {X 0.006,Y -431.154,Z 1341.523,A 0.000,B 0.000,C 90.000,E1 274.131} C_DIS
LIN {X -0.093,Y -424.843,Z 1341.521,A 0.000,B 0.000,C 90.000,E1 273.726} C_DIS
LIN {X 0.141,Y -418.388,Z 1341.519,A 0.000,B 0.000,C 90.000,E1 273.326} C_DIS
LIN {X -0.131,Y -411.777,Z 1341.517,A 0.000,B 0.000,C 90.000,E1 273.037} C_DIS
LIN {X -0.148,Y -405.235,Z 1341.515,A 0.000,B 0.000,C 90.000,E1 272.751} C_DIS
LIN {X 0.062,Y -394.452,Z 1341.513,A 0.000,B 0.000,C 90.000,E1 272.350} C_DIS
LIN {X -0.102,Y -387.359,Z 1341.512,A 0.000,B 0.000,C 90.000,E1 272.178} C_DIS
LIN {X -0.165,Y -375.839,Z 1341.511,A 0.000,B 0.000,C 90.000,E1 271.949} C_DIS
LIN {X 0.154,Y -366.656,Z 1341.510,A 0.000,B 0.000,C 90.000,E1 271.776} C_DIS
LIN {X 0.161,Y -352.642,Z 1341.509,A 0.000,B 0.000,C 90.000,E1 271.661} C_DIS
LIN {X 0.046,Y -348.426,Z 1341.509,A 0.000,B 0.000,C 90.000,E1 271.661} C_DIS
LIN {X -0.010,Y -339.953,Z 1341.509,A 0.000,B 0.000,C 90.000,E1 271.661} C_DIS
LIN {X -0.035,Y -181.322,Z 1341.509,A 0.000,B 0.000,C 90.000,E1 271.661} C_DIS
LIN {X 0.010,Y -181.574,Z 1341.501,A 0.000,B 0.000,C 90.000,E1 270.115} C_DIS
LIN {X -0.033,Y -180.906,Z 1341.474,A 0.000,B 0.000,C 90.000,E1 265.412} C_DIS
LIN {X 0.041,Y -180.705,Z 1341.470,A 0.000,B 0.000,C 90.000,E1 264.546} C_DIS
LIN {X -0.057,Y -178.791,Z 1341.442,A 0.000,B 0.000,C 90.000,E1 259.511} C_DIS
LIN {X 0.020,Y -175.837,Z 1341.413,A 0.000,B 0.000,C 90.000,E1 254.393} C_DIS
LIN {X 0.020,Y -172.027,Z 1341.385,A 0.000,B 0.000,C 90.000,E1 249.263} C_DIS
LIN {X -0.004,Y -171.453,Z 1341.380,A 0.000,B 0.000,C 90.000,E1 248.411} C_DIS
LIN {X -0.023,Y -167.687,Z 1341.356,A 0.000,B 0.000,C 90.000,E1 244.101} C_DIS
LIN {X -0.010,Y -166.366,Z 1341.346,A 0.000,B 0.000,C 90.000,E1 242.359} C_DIS
LIN {X -0.017,Y -163.098,Z 1341.327,A 0.000,B 0.000,C 90.000,E1 238.869} C_DIS
LIN {X 0.033,Y -161.043,Z 1341.312,A 0.000,B 0.000,C 90.000,E1 236.215} C_DIS
LIN {X 0.017,Y -157.780,Z 1341.293,A 0.000,B 0.000,C 90.000,E1 232.683} C_DIS
LIN {X 0.080,Y -155.817,Z 1341.278,A 0.000,B 0.000,C 90.000,E1 229.989} C_DIS
LIN {X -0.082,Y -152.069,Z 1341.253,A 0.000,B 0.000,C 90.000,E1 225.567} C_DIS
LIN {X -0.062,Y -150.319,Z 1341.238,A 0.000,B 0.000,C 90.000,E1 222.852} C_DIS
LIN {X -0.041,Y -147.061,Z 1341.213,A 0.000,B 0.000,C 90.000,E1 218.302} C_DIS
LIN {X 0.067,Y -145.638,Z 1341.198,A 0.000,B 0.000,C 90.000,E1 215.518} C_DIS
LIN {X 0.064,Y -143.021,Z 1341.172,A 0.000,B 0.000,C 90.000,E1 210.924} C_DIS
LIN {X -0.005,Y -141.647,Z 1341.151,A 0.000,B 0.000,C 90.000,E1 207.257} C_DIS
LIN {X 0.045,Y -139.442,Z 1341.115,A 0.000,B 0.000,C 90.000,E1 200.737} C_DIS
LIN {X -0.033,Y -139.175,Z 1341.105,A 0.000,B 0.000,C 90.000,E1 198.906} C_DIS
LIN {X -0.004,Y -138.319,Z 1341.053,A 0.000,B 0.000,C 90.000,E1 189.557} C_DIS
LIN {X 0.005,Y -139.470,Z 1341.006,A 0.000,B 0.000,C 90.000,E1 181.146} C_DIS
LIN {X -0.055,Y -141.040,Z 1340.975,A 0.000,B 0.000,C 90.000,E1 175.584} C_DIS
LIN {X 0.040,Y -142.409,Z 1340.960,A 0.000,B 0.000,C 90.000,E1 172.761} C_DIS
LIN {X -0.039,Y -144.642,Z 1340.934,A 0.000,B 0.000,C 90.000,E1 168.173} C_DIS
LIN {X 0.021,Y -147.838,Z 1340.909,A 0.000,B 0.000,C 90.000,E1 163.559} C_DIS
LIN {X -0.035,Y -150.536,Z 1340.888,A 0.000,B 0.000,C 90.000,E1 159.934} C_DIS
LIN {X -0.016,Y -154.000,Z 1340.868,A 0.000,B 0.000,C 90.000,E1 156.305} C_DIS
LIN {X 0.044,Y -157.414,Z 1340.848,A 0.000,B 0.000,C 90.000,E1 152.692} C_DIS
LIN {X 0.066,Y -161.624,Z 1340.829,A 0.000,B 0.000,C 90.000,E1 149.125} C_DIS
LIN {X 0.085,Y -165.820,Z 1340.809,A 0.000,B 0.000,C 90.000,E1 145.595} C_DIS
LIN {X 0.078,Y -170.788,Z 1340.790,A 0.000,B 0.000,C 90.000,E1 142.110} C_DIS
LIN {X -0.005,Y -175.659,Z 1340.771,A 0.000,B 0.000,C 90.000,E1 138.690} C_DIS
LIN {X -0.007,Y -181.273,Z 1340.752,A 0.000,B 0.000,C 90.000,E1 135.283} C_DIS
LIN {X -0.007,Y -186.749,Z 1340.733,A 0.000,B 0.000,C 90.000,E1 131.919} C_DIS
LIN {X -0.057,Y -191.345,Z 1340.719,A 0.000,B 0.000,C 90.000,E1 129.439} C_DIS
LIN {X -0.011,Y -197.181,Z 1340.701,A 0.000,B 0.000,C 90.000,E1 126.137} C_DIS
LIN {X 0.049,Y -199.195,Z 1340.695,A 0.000,B 0.000,C 90.000,E1 125.105} C_DIS
LIN {X 0.041,Y -309.307,Z 1340.695,A 0.000,B 0.000,C 90.000,E1 125.105} C_DIS
LIN {X 0.209,Y -311.595,Z 1340.695,A 0.000,B 0.000,C 90.000,E1 125.025} C_DIS
LIN {X 0.073,Y -316.537,Z 1340.693,A 0.000,B 0.000,C 90.000,E1 124.771} C_DIS
LIN {X 0.116,Y -319.313,Z 1340.692,A 0.000,B 0.000,C 90.000,E1 124.485} C_DIS
LIN {X 0.180,Y -322.956,Z 1340.689,A 0.000,B 0.000,C 90.000,E1 123.913} C_DIS
LIN {X -0.011,Y -324.394,Z 1340.687,A 0.000,B 0.000,C 90.000,E1 123.627} C_DIS
LIN {X 0.187,Y -337.198,Z 1340.668,A 0.000,B 0.000,C 90.000,E1 120.129} C_DIS
LIN {X 0.002,Y -349.114,Z 1340.652,A 0.000,B 0.000,C 90.000,E1 117.385} C_DIS
LIN {X 0.146,Y -362.488,Z 1340.637,A 0.000,B 0.000,C 90.000,E1 114.643} C_DIS
LIN {X 0.128,Y -375.691,Z 1340.624,A 0.000,B 0.000,C 90.000,E1 112.280} C_DIS
LIN {X -0.060,Y -390.226,Z 1340.611,A 0.000,B 0.000,C 90.000,E1 109.993} C_DIS
LIN {X 0.206,Y -406.197,Z 1340.599,A 0.000,B 0.000,C 90.000,E1 107.692} C_DIS
LIN {X 0.247,Y -423.714,Z 1340.586,A 0.000,B 0.000,C 90.000,E1 105.481} C_DIS
LIN {X 0.104,Y -442.872,Z 1340.574,A 0.000,B 0.000,C 90.000,E1 103.355} C_DIS
LIN {X -0.014,Y -462.968,Z 1340.563,A 0.000,B 0.000,C 90.000,E1 101.366} C_DIS
LIN {X 0.167,Y -480.788,Z 1340.554,A 0.000,B 0.000,C 90.000,E1 99.726} C_DIS
LIN {X 0.192,Y -482.608,Z 1340.553,A 0.000,B 0.000,C 90.000,E1 99.500} C_DIS
LIN {X 0.075,Y -484.157,Z 1340.552,A 0.000,B 0.000,C 90.000,E1 99.265} C_DIS
LIN {X -0.045,Y -485.314,Z 1340.550,A 0.000,B 0.000,C 90.000,E1 99.029} C_DIS
LIN {X 0.139,Y -486.698,Z 1340.547,A 0.000,B 0.000,C 90.000,E1 98.511} C_DIS
LIN {X -0.150,Y -487.044,Z 1340.545,A 0.000,B 0.000,C 90.000,E1 98.049} C_DIS
LIN {X 0.053,Y -486.409,Z 1340.542,A 0.000,B 0.000,C 90.000,E1 97.530} C_DIS
LIN {X -0.223,Y -484.689,Z 1340.539,A 0.000,B 0.000,C 90.000,E1 97.068} C_DIS
LIN {X 0.147,Y -483.324,Z 1340.538,A 0.000,B 0.000,C 90.000,E1 96.777} C_DIS
LIN {X -0.208,Y -469.095,Z 1340.527,A 0.000,B 0.000,C 90.000,E1 94.821} C_DIS
LIN {X -0.174,Y -457.410,Z 1340.517,A 0.000,B 0.000,C 90.000,E1 93.037} C_DIS
LIN {X -0.043,Y -442.534,Z 1340.504,A 0.000,B 0.000,C 90.000,E1 90.688} C_DIS
LIN {X 0.006,Y -426.162,Z 1340.488,A 0.000,B 0.000,C 90.000,E1 87.764} C_DIS
LIN {X 0.022,Y -416.035,Z 1340.477,A 0.000,B 0.000,C 90.000,E1 85.869} C_DIS
LIN {X 0.167,Y -407.220,Z 1340.468,A 0.000,B 0.000,C 90.000,E1 84.204} C_DIS
LIN {X -0.129,Y -396.741,Z 1340.457,A 0.000,B 0.000,C 90.000,E1 82.299} C_DIS
LIN {X 0.140,Y -387.475,Z 1340.448,A 0.000,B 0.000,C 90.000,E1 80.566} C_DIS
LIN {X -0.013,Y -378.042,Z 1340.438,A 0.000,B 0.000,C 90.000,E1 78.870} C_DIS
LIN {X 0.041,Y -368.343,Z 1340.428,A 0.000,B 0.000,C 90.000,E1 77.117} C_DIS
LIN {X 0.041,Y -356.808,Z 1340.417,A 0.000,B 0.000,C 90.000,E1 75.046} C_DIS
LIN {X -0.123,Y -346.964,Z 1340.407,A 0.000,B 0.000,C 90.000,E1 73.268} C_DIS
LIN {X 0.059,Y -335.292,Z 1340.395,A 0.000,B 0.000,C 90.000,E1 71.094} C_DIS
LIN {X 0.052,Y -322.196,Z 1340.381,A 0.000,B 0.000,C 90.000,E1 68.592} C_DIS
LIN {X 0.101,Y -305.222,Z 1340.361,A 0.000,B 0.000,C 90.000,E1 65.049} C_DIS
LIN {X -0.163,Y -296.796,Z 1340.351,A 0.000,B 0.000,C 90.000,E1 63.127} C_DIS
LIN {X -0.034,Y -289.155,Z 1340.339,A 0.000,B 0.000,C 90.000,E1 61.101} C_DIS
LIN {X -0.081,Y -281.240,Z 1340.326,A 0.000,B 0.000,C 90.000,E1 58.742} C_DIS
LIN {X -0.101,Y -271.188,Z 1340.307,A 0.000,B 0.000,C 90.000,E1 55.308} C_DIS
LIN {X 0.027,Y -261.902,Z 1340.288,A 0.000,B 0.000,C 90.000,E1 51.778} C_DIS
LIN {X -0.105,Y -253.175,Z 1340.268,A 0.000,B 0.000,C 90.000,E1 48.243} C_DIS
LIN {X -0.008,Y -244.930,Z 1340.248,A 0.000,B 0.000,C 90.000,E1 44.595} C_DIS
LIN {X 0.007,Y -237.313,Z 1340.227,A 0.000,B 0.000,C 90.000,E1 40.906} C_DIS
LIN {X 0.038,Y -230.479,Z 1340.206,A 0.000,B 0.000,C 90.000,E1 37.156} C_DIS
LIN {X 0.002,Y -224.527,Z 1340.185,A 0.000,B 0.000,C 90.000,E1 33.372} C_DIS
LIN {X -0.018,Y -219.637,Z 1340.164,A 0.000,B 0.000,C 90.000,E1 29.539} C_DIS
LIN {X -0.079,Y -215.058,Z 1340.138,A 0.000,B 0.000,C 90.000,E1 24.899} C_DIS
LIN {X -0.025,Y -212.010,Z 1340.116,A 0.000,B 0.000,C 90.000,E1 20.972} C_DIS
LIN {X -0.046,Y -209.288,Z 1340.095,A 0.000,B 0.000,C 90.000,E1 17.040} C_DIS
LIN {X -0.084,Y -207.283,Z 1340.077,A 0.000,B 0.000,C 90.000,E1 13.883} C_DIS
LIN {X 0.075,Y -205.303,Z 1340.059,A 0.000,B 0.000,C 90.000,E1 10.658} C_DIS
LIN {X 0.077,Y -203.222,Z 1340.037,A 0.000,B 0.000,C 90.000,E1 6.663} C_DIS
LIN {X 0.000,Y -200.859,Z 1340.000,A 0.000,B 0.000,C 90.000,E1 360.000} C_DIS
LIN {X -0.105,Y -200.323,Z 1339.970,A 0.000,B 0.000,C 90.000,E1 354.723} C_DIS
LIN {X -0.057,Y -201.856,Z 1339.926,A 0.000,B 0.000,C 90.000,E1 346.645} C_DIS
LIN {X -0.112,Y -204.881,Z 1339.895,A 0.000,B 0.000,C 90.000,E1 341.040} C_DIS
LIN {X -0.018,Y -208.925,Z 1339.868,A 0.000,B 0.000,C 90.000,E1 336.230} C_DIS
LIN {X -0.034,Y -213.440,Z 1339.846,A 0.000,B 0.000,C 90.000,E1 332.281} C_DIS
LIN {X 0.118,Y -218.963,Z 1339.824,A 0.000,B 0.000,C 90.000,E1 328.329} C_DIS
LIN {X 0.048,Y -225.617,Z 1339.803,A 0.000,B 0.000,C 90.000,E1 324.482} C_DIS
LIN {X -0.060,Y -231.769,Z 1339.786,A 0.000,B 0.000,C 90.000,E1 321.457} C_DIS
LIN {X 0.022,Y -240.407,Z 1339.765,A 0.000,B 0.000,C 90.000,E1 317.676} C_DIS
LIN {X 0.022,Y -249.274,Z 1339.746,A 0.000,B 0.000,C 90.000,E1 314.352} C_DIS
LIN {X -0.102,Y -257.085,Z 1339.732,A 0.000,B 0.000,C 90.000,E1 311.838} C_DIS
LIN {X -0.035,Y -265.938,Z 1339.718,A 0.000,B 0.000,C 90.000,E1 309.322} C_DIS
LIN {X -0.154,Y -274.388,Z 1339.707,A 0.000,B 0.000,C 90.000,E1 307.237} C_DIS
LIN {X -0.160,Y -285.359,Z 1339.693,A 0.000,B 0.000,C 90.000,E1 304.818} C_DIS
LIN {X 0.020,Y -294.134,Z 1339.684,A 0.000,B 0.000,C 90.000,E1 303.086} C_DIS
LIN {X 0.025,Y -303.850,Z 1339.675,A 0.000,B 0.000,C 90.000,E1 301.416} C_DIS
LIN {X -0.122,Y -312.369,Z 1339.667,A 0.000,B 0.000,C 90.000,E1 300.129} C_DIS
LIN {X 0.108,Y -326.688,Z 1339.656,A 0.000,B 0.000,C 90.000,E1 298.153} C_DIS
LIN {X -0.012,Y -347.484,Z 1339.643,A 0.000,B 0.000,C 90.000,E1 295.720} C_DIS
LIN {X 0.115,Y -360.700,Z 1339.635,A 0.000,B 0.000,C 90.000,E1 294.207} C_DIS
LIN {X -0.075,Y -373.692,Z 1339.626,A 0.000,B 0.000,C 90.000,E1 292.770} C_DIS
LIN {X 0.088,Y -383.748,Z 1339.620,A 0.000,B 0.000,C 90.000,E1 291.589} C_DIS
LIN {X -0.041,Y -395.966,Z 1339.612,A 0.000,B 0.000,C 90.000,E1 290.174} C_DIS
LIN {X 0.166,Y -413.208,Z 1339.601,A 0.000,B 0.000,C 90.000,E1 288.181} C_DIS
LIN {X 0.083,Y -422.848,Z 1339.595,A 0.000,B 0.000,C 90.000,E1 287.094} C_DIS
LIN {X -0.014,Y -431.980,Z 1339.589,A 0.000,B 0.000,C 90.000,E1 286.024} C_DIS
LIN {X -0.195,Y -438.256,Z 1339.585,A 0.000,B 0.000,C 90.000,E1 285.245} C_DIS
LIN {X -0.013,Y -443.876,Z 1339.580,A 0.000,B 0.000,C 90.000,E1 284.426} C_DIS
LIN {X -0.094,Y -448.852,Z 1339.576,A 0.000,B 0.000,C 90.000,E1 283.647} C_DIS
LIN {X 0.193,Y -453.017,Z 1339.571,A 0.000,B 0.000,C 90.000,E1 282.827} C_DIS
LIN {X -0.181,Y -455.326,Z 1339.568,A 0.000,B 0.000,C 90.000,E1 282.355} C_DIS
LIN {X -0.098,Y -457.318,Z 1339.566,A 0.000,B 0.000,C 90.000,E1 281.827} C_DIS
LIN {X -0.008,Y -458.966,Z 1339.563,A 0.000,B 0.000,C 90.000,E1 281.299} C_DIS
LIN {X 0.004,Y -460.295,Z 1339.560,A 0.000,B 0.000,C 90.000,E1 280.782} C_DIS
LIN {X 0.116,Y -461.140,Z 1339.557,A 0.000,B 0.000,C 90.000,E1 280.254} C_DIS
LIN {X 0.232,Y -461.662,Z 1339.554,A 0.000,B 0.000,C 90.000,E1 279.726} C_DIS
LIN {X -0.180,Y -461.723,Z 1339.551,A 0.000,B 0.000,C 90.000,E1 279.265} C_DIS
LIN {X -0.131,Y -461.255,Z 1339.548,A 0.000,B 0.000,C 90.000,E1 278.746} C_DIS
LIN {X -0.012,Y -460.335,Z 1339.546,A 0.000,B 0.000,C 90.000,E1 278.219} C_DIS
LIN {X 0.036,Y -458.921,Z 1339.543,A 0.000,B 0.000,C 90.000,E1 277.701} C_DIS
LIN {X 0.081,Y -456.990,Z 1339.540,A 0.000,B 0.000,C 90.000,E1 277.182} C_DIS
LIN {X 0.118,Y -454.483,Z 1339.537,A 0.000,B 0.000,C 90.000,E1 276.663} C_DIS
LIN {X 0.137,Y -451.418,Z 1339.534,A 0.000,B 0.000,C 90.000,E1 276.144} C_DIS
LIN {X 0.138,Y -447.736,Z 1339.531,A 0.000,B 0.000,C 90.000,E1 275.625} C_DIS
LIN {X 0.120,Y -443.272,Z 1339.528,A 0.000,B 0.000,C 90.000,E1 275.106} C_DIS
LIN {X 0.077,Y -437.777,Z 1339.526,A 0.000,B 0.000,C 90.000,E1 274.588} C_DIS
LIN {X -0.094,Y -431.693,Z 1339.523,A 0.000,B 0.000,C 90.000,E1 274.131} C_DIS
LIN {X -0.205,Y -425.519,Z 1339.521,A 0.000,B 0.000,C 90.000,E1 273.726} C_DIS
LIN {X -0.029,Y -418.856,Z 1339.518,A 0.000,B 0.000,C 90.000,E1 273.326} C_DIS
LIN {X -0.091,Y -409.230,Z 1339.516,A 0.000,B 0.000,C 90.000,E1 272.865} C_DIS
LIN {X 0.026,Y -402.536,Z 1339.514,A 0.000,B 0.000,C 90.000,E1 272.579} C_DIS
LIN {X -0.013,Y -395.616,Z 1339.513,A 0.000,B 0.000,C 90.000,E1 272.350} C_DIS
LIN {X 0.176,Y -388.394,Z 1339.512,A 0.000,B 0.000,C 90.000,E1 272.121} C_DIS
LIN {X -0.164,Y -381.004,Z 1339.511,A 0.000,B 0.000,C 90.000,E1 272.007} C_DIS
LIN {X 0.076,Y -372.936,Z 1339.510,A 0.000,B 0.000,C 90.000,E1 271.835} C_DIS
LIN {X 0.117,Y -363.746,Z 1339.510,A 0.000,B 0.000,C 90.000,E1 271.718} C_DIS
LIN {X -0.064,Y -351.147,Z 1339.509,A 0.000,B 0.000,C 90.000,E1 271.661} C_DIS
LIN {X -0.120,Y -347.100,Z 1339.509,A 0.000,B 0.000,C 90.000,E1 271.661} C_DIS
LIN {X 0.089,Y -181.326,Z 1339.509,A 0.000,B 0.000,C 90.000,E1 271.604} C_DIS
LIN {X -0.047,Y -181.573,Z 1339.501,A 0.000,B 0.000,C 90.000,E1 270.115} C_DIS
LIN {X -0.090,Y -180.906,Z 1339.474,A 0.000,B 0.000,C 90.000,E1 265.412} C_DIS
LIN {X -0.016,Y -180.697,Z 1339.470,A 0.000,B 0.000,C 90.000,E1 264.546} C_DIS
LIN {X 0.063,Y -178.781,Z 1339.442,A 0.000,B 0.000,C 90.000,E1 259.454} C_DIS
LIN {X -0.035,Y -175.827,Z 1339.413,A 0.000,B 0.000,C 90.000,E1 254.393} C_DIS
LIN {X -0.035,Y -172.015,Z 1339.385,A 0.000,B 0.000,C 90.000,E1 249.263} C_DIS
LIN {X -0.059,Y -171.437,Z 1339.380,A 0.000,B 0.000,C 90.000,E1 248.411} C_DIS
LIN {X -0.004,Y -167.673,Z 1339.356,A 0.000,B 0.000,C 90.000,E1 244.076} C_DIS
LIN {X -0.064,Y -166.347,Z 1339.346,A 0.000,B 0.000,C 90.000,E1 242.359} C_DIS
LIN {X -0.071,Y -163.082,Z 1339.327,A 0.000,B 0.000,C 90.000,E1 238.869} C_DIS
LIN {X -0.020,Y -161.024,Z 1339.312,A 0.000,B 0.000,C 90.000,E1 236.215} C_DIS
LIN {X -0.035,Y -157.765,Z 1339.293,A 0.000,B 0.000,C 90.000,E1 232.683} C_DIS
LIN {X 0.027,Y -155.803,Z 1339.278,A 0.000,B 0.000,C 90.000,E1 229.989} C_DIS
LIN {X 0.082,Y -152.055,Z 1339.253,A 0.000,B 0.000,C 90.000,E1 225.486} C_DIS
LIN {X -0.011,Y -150.304,Z 1339.238,A 0.000,B 0.000,C 90.000,E1 222.813} C_DIS
LIN {X 0.025,Y -147.049,Z 1339.213,A 0.000,B 0.000,C 90.000,E1 218.257} C_DIS
LIN {X 0.017,Y -145.628,Z 1339.197,A 0.000,B 0.000,C 90.000,E1 215.518} C_DIS
LIN {X 0.015,Y -143.012,Z 1339.172,A 0.000,B 0.000,C 90.000,E1 210.924} C_DIS
LIN {X -0.053,Y -141.638,Z 1339.151,A 0.000,B 0.000,C 90.000,E1 207.257} C_DIS
LIN {X -0.003,Y -139.439,Z 1339.115,A 0.000,B 0.000,C 90.000,E1 200.737} C_DIS
LIN {X 0.051,Y -139.171,Z 1339.105,A 0.000,B 0.000,C 90.000,E1 198.852} C_DIS
LIN {X -0.052,Y -138.317,Z 1339.053,A 0.000,B 0.000,C 90.000,E1 189.557} C_DIS
LIN {X -0.043,Y -139.473,Z 1339.006,A 0.000,B 0.000,C 90.000,E1 181.146} C_DIS
LIN {X 0.037,Y -141.049,Z 1338.975,A 0.000,B 0.000,C 90.000,E1 175.527} C_DIS
LIN {X -0.009,Y -142.419,Z 1338.960,A 0.000,B 0.000,C 90.000,E1 172.761} C_DIS
LIN {X 0.053,Y -144.655,Z 1338.934,A 0.000,B 0.000,C 90.000,E1 168.117} C_DIS
LIN {X -0.030,Y -147.851,Z 1338.909,A 0.000,B 0.000,C 90.000,E1 163.559} C_DIS
LIN {X 0.056,Y -150.552,Z 1338.888,A 0.000,B 0.000,C 90.000,E1 159.880} C_DIS
LIN {X -0.067,Y -154.019,Z 1338.868,A 0.000,B 0.000,C 90.000,E1 156.305} C_DIS
LIN {X -0.009,Y -157.434,Z 1338.848,A 0.000,B 0.000,C 90.000,E1 152.692} C_DIS
LIN {X 0.013,Y -161.648,Z 1338.828,A 0.000,B 0.000,C 90.000,E1 149.125} C_DIS
LIN {X 0.030,Y -165.844,Z 1338.809,A 0.000,B 0.000,C 90.000,E1 145.595} C_DIS
LIN {X 0.023,Y -170.817,Z 1338.790,A 0.000,B 0.000,C 90.000,E1 142.110} C_DIS
LIN {X -0.061,Y -175.687,Z 1338.770,A 0.000,B 0.000,C 90.000,E1 138.690} C_DIS
LIN {X 0.062,Y -181.300,Z 1338.751,A 0.000,B 0.000,C 90.000,E1 135.243} C_DIS
LIN {X -0.065,Y -186.781,Z 1338.733,A 0.000,B 0.000,C 90.000,E1 131.919} C_DIS
LIN {X 0.006,Y -191.373,Z 1338.719,A 0.000,B 0.000,C 90.000,E1 129.402} C_DIS
LIN {X 0.088,Y -197.214,Z 1338.701,A 0.000,B 0.000,C 90.000,E1 126.091} C_DIS
LIN {X 0.076,Y -199.180,Z 1338.695,A 0.000,B 0.000,C 90.000,E1 125.105} C_DIS
LIN {X 0.068,Y -308.613,Z 1338.695,A 0.000,B 0.000,C 90.000,E1 125.105} C_DIS
LIN {X 0.018,Y -309.608,Z 1338.695,A 0.000,B 0.000,C 90.000,E1 125.105} C_DIS
LIN {X 0.045,Y -314.079,Z 1338.694,A 0.000,B 0.000,C 90.000,E1 124.945} C_DIS
LIN {X -0.111,Y -316.348,Z 1338.693,A 0.000,B 0.000,C 90.000,E1 124.818} C_DIS
LIN {X 0.020,Y -319.435,Z 1338.692,A 0.000,B 0.000,C 90.000,E1 124.485} C_DIS
LIN {X 0.084,Y -323.021,Z 1338.688,A 0.000,B 0.000,C 90.000,E1 123.913} C_DIS
LIN {X -0.106,Y -324.440,Z 1338.687,A 0.000,B 0.000,C 90.000,E1 123.627} C_DIS
LIN {X 0.089,Y -337.243,Z 1338.667,A 0.000,B 0.000,C 90.000,E1 120.129} C_DIS
LIN {X -0.097,Y -349.167,Z 1338.652,A 0.000,B 0.000,C 90.000,E1 117.385} C_DIS
LIN {X 0.043,Y -362.550,Z 1338.637,A 0.000,B 0.000,C 90.000,E1 114.643} C_DIS
LIN {X 0.023,Y -375.761,Z 1338.624,A 0.000,B 0.000,C 90.000,E1 112.280} C_DIS
LIN {X -0.167,Y -390.306,Z 1338.611,A 0.000,B 0.000,C 90.000,E1 109.993} C_DIS
LIN {X 0.098,Y -406.286,Z 1338.598,A 0.000,B 0.000,C 90.000,E1 107.692} C_DIS
LIN {X 0.136,Y -423.814,Z 1338.586,A 0.000,B 0.000,C 90.000,E1 105.481} C_DIS
LIN {X -0.007,Y -442.982,Z 1338.574,A 0.000,B 0.000,C 90.000,E1 103.355} C_DIS
LIN {X -0.124,Y -463.082,Z 1338.563,A 0.000,B 0.000,C 90.000,E1 101.366} C_DIS
LIN {X -0.046,Y -478.511,Z 1338.555,A 0.000,B 0.000,C 90.000,E1 99.962} C_DIS
LIN {X 0.061,Y -480.852,Z 1338.554,A 0.000,B 0.000,C 90.000,E1 99.726} C_DIS
LIN {X 0.087,Y -482.623,Z 1338.553,A 0.000,B 0.000,C 90.000,E1 99.500} C_DIS
LIN {X -0.031,Y -484.132,Z 1338.551,A 0.000,B 0.000,C 90.000,E1 99.265} C_DIS
LIN {X -0.150,Y -485.258,Z 1338.550,A 0.000,B 0.000,C 90.000,E1 99.029} C_DIS
LIN {X 0.033,Y -486.592,Z 1338.547,A 0.000,B 0.000,C 90.000,E1 98.511} C_DIS
LIN {X 0.226,Y -486.894,Z 1338.545,A 0.000,B 0.000,C 90.000,E1 97.992} C_DIS
LIN {X -0.054,Y -486.213,Z 1338.542,A 0.000,B 0.000,C 90.000,E1 97.530} C_DIS
LIN {X 0.151,Y -484.441,Z 1338.539,A 0.000,B 0.000,C 90.000,E1 97.011} C_DIS
LIN {X 0.040,Y -483.041,Z 1338.538,A 0.000,B 0.000,C 90.000,E1 96.777} C_DIS
LIN {X 0.188,Y -468.798,Z 1338.527,A 0.000,B 0.000,C 90.000,E1 94.759} C_DIS
LIN {X 0.168,Y -457.086,Z 1338.517,A 0.000,B 0.000,C 90.000,E1 92.980} C_DIS
LIN {X -0.162,Y -442.241,Z 1338.504,A 0.000,B 0.000,C 90.000,E1 90.688} C_DIS
LIN {X -0.117,Y -425.857,Z 1338.488,A 0.000,B 0.000,C 90.000,E1 87.764} C_DIS
LIN {X -0.105,Y -415.739,Z 1338.477,A 0.000,B 0.000,C 90.000,E1 85.869} C_DIS
LIN {X 0.039,Y -406.920,Z 1338.468,A 0.000,B 0.000,C 90.000,E1 84.204} C_DIS
LIN {X 0.132,Y -396.474,Z 1338.457,A 0.000,B 0.000,C 90.000,E1 82.243} C_DIS
LIN {X 0.070,Y -387.185,Z 1338.448,A 0.000,B 0.000,C 90.000,E1 80.557} C_DIS
LIN {X -0.148,Y -377.758,Z 1338.438,A 0.000,B 0.000,C 90.000,E1 78.870} C_DIS
LIN {X -0.096,Y -368.058,Z 1338.428,A 0.000,B 0.000,C 90.000,E1 77.117} C_DIS
LIN {X -0.098,Y -356.517,Z 1338.417,A 0.000,B 0.000,C 90.000,E1 75.046} C_DIS
LIN {X 0.169,Y -346.673,Z 1338.407,A 0.000,B 0.000,C 90.000,E1 73.196} C_DIS
LIN {X -0.083,Y -335.008,Z 1338.395,A 0.000,B 0.000,C 90.000,E1 71.094} C_DIS
LIN {X -0.091,Y -321.933,Z 1338.381,A 0.000,B 0.000,C 90.000,E1 68.592} C_DIS
LIN {X -0.043,Y -304.967,Z 1338.361,A 0.000,B 0.000,C 90.000,E1 65.049} C_DIS
LIN {X -0.032,Y -295.220,Z 1338.349,A 0.000,B 0.000,C 90.000,E1 62.743} C_DIS
LIN {X 0.045,Y -286.602,Z 1338.336,A 0.000,B 0.000,C 90.000,E1 60.383} C_DIS
LIN {X 0.006,Y -276.920,Z 1338.318,A 0.000,B 0.000,C 90.000,E1 57.327} C_DIS
LIN {X -0.003,Y -267.269,Z 1338.299,A 0.000,B 0.000,C 90.000,E1 53.863} C_DIS
LIN {X -0.100,Y -258.215,Z 1338.280,A 0.000,B 0.000,C 90.000,E1 50.356} C_DIS
LIN {X -0.026,Y -251.433,Z 1338.264,A 0.000,B 0.000,C 90.000,E1 47.472} C_DIS
LIN {X 0.014,Y -243.320,Z 1338.244,A 0.000,B 0.000,C 90.000,E1 43.824} C_DIS
LIN {X -0.021,Y -235.853,Z 1338.223,A 0.000,B 0.000,C 90.000,E1 40.135} C_DIS
LIN {X 0.002,Y -229.200,Z 1338.202,A 0.000,B 0.000,C 90.000,E1 36.377} C_DIS
LIN {X 0.113,Y -223.442,Z 1338.181,A 0.000,B 0.000,C 90.000,E1 32.546} C_DIS
LIN {X -0.058,Y -218.798,Z 1338.160,A 0.000,B 0.000,C 90.000,E1 28.743} C_DIS
LIN {X -0.056,Y -214.398,Z 1338.134,A 0.000,B 0.000,C 90.000,E1 24.079} C_DIS
LIN {X 0.093,Y -211.405,Z 1338.112,A 0.000,B 0.000,C 90.000,E1 20.120} C_DIS
LIN {X -0.011,Y -208.727,Z 1338.090,A 0.000,B 0.000,C 90.000,E1 16.205} C_DIS
LIN {X 0.086,Y -206.704,Z 1338.072,A 0.000,B 0.000,C 90.000,E1 13.008} C_DIS
LIN {X 0.106,Y -203.873,Z 1338.046,A 0.000,B 0.000,C 90.000,E1 8.219} C_DIS
LIN {X -0.005,Y -201.741,Z 1338.019,A 0.000,B 0.000,C 90.000,E1 3.440} C_DIS
LIN {X -0.078,Y -200.370,Z 1337.984,A 0.000,B 0.000,C 90.000,E1 357.135} C_DIS
LIN {X -0.019,Y -201.060,Z 1337.939,A 0.000,B 0.000,C 90.000,E1 349.050} C_DIS
LIN {X 0.041,Y -203.893,Z 1337.903,A 0.000,B 0.000,C 90.000,E1 342.598} C_DIS
LIN {X 0.073,Y -207.490,Z 1337.877,A 0.000,B 0.000,C 90.000,E1 337.794} C_DIS
LIN {X 0.016,Y -211.635,Z 1337.855,A 0.000,B 0.000,C 90.000,E1 333.845} C_DIS
LIN {X -0.001,Y -216.740,Z 1337.833,A 0.000,B 0.000,C 90.000,E1 329.921} C_DIS
LIN {X 0.113,Y -222.977,Z 1337.811,A 0.000,B 0.000,C 90.000,E1 326.008} C_DIS
LIN {X 0.059,Y -230.262,Z 1337.790,A 0.000,B 0.000,C 90.000,E1 322.190} C_DIS
LIN {X -0.060,Y -238.728,Z 1337.769,A 0.000,B 0.000,C 90.000,E1 318.447} C_DIS
LIN {X 0.058,Y -247.324,Z 1337.750,A 0.000,B 0.000,C 90.000,E1 315.081} C_DIS
LIN {X 0.062,Y -254.846,Z 1337.736,A 0.000,B 0.000,C 90.000,E1 312.528} C_DIS
LIN {X 0.086,Y -263.384,Z 1337.722,A 0.000,B 0.000,C 90.000,E1 310.011} C_DIS
LIN {X -0.047,Y -273.009,Z 1337.709,A 0.000,B 0.000,C 90.000,E1 307.569} C_DIS
LIN {X -0.082,Y -283.815,Z 1337.695,A 0.000,B 0.000,C 90.000,E1 305.152} C_DIS
LIN {X 0.052,Y -294.253,Z 1337.684,A 0.000,B 0.000,C 90.000,E1 303.086} C_DIS
LIN {X 0.059,Y -303.962,Z 1337.675,A 0.000,B 0.000,C 90.000,E1 301.416} C_DIS
LIN {X -0.084,Y -312.496,Z 1337.667,A 0.000,B 0.000,C 90.000,E1 300.129} C_DIS
LIN {X -0.004,Y -326.780,Z 1337.656,A 0.000,B 0.000,C 90.000,E1 298.180} C_DIS
LIN {X 0.101,Y -347.885,Z 1337.643,A 0.000,B 0.000,C 90.000,E1 295.668} C_DIS
LIN {X -0.017,Y -360.974,Z 1337.635,A 0.000,B 0.000,C 90.000,E1 294.207} C_DIS
LIN {X -0.144,Y -373.843,Z 1337.626,A 0.000,B 0.000,C 90.000,E1 292.770} C_DIS
LIN {X 0.012,Y -383.890,Z 1337.620,A 0.000,B 0.000,C 90.000,E1 291.589} C_DIS
LIN {X -0.085,Y -398.540,Z 1337.610,A 0.000,B 0.000,C 90.000,E1 289.885} C_DIS
LIN {X 0.091,Y -413.332,Z 1337.601,A 0.000,B 0.000,C 90.000,E1 288.181} C_DIS
LIN {X 0.005,Y -422.980,Z 1337.595,A 0.000,B 0.000,C 90.000,E1 287.094} C_DIS
LIN {X -0.091,Y -432.109,Z 1337.589,A 0.000,B 0.000,C 90.000,E1 286.024} C_DIS
LIN {X 0.152,Y -438.392,Z 1337.584,A 0.000,B 0.000,C 90.000,E1 285.190} C_DIS
LIN {X 0.129,Y -442.254,Z 1337.582,A 0.000,B 0.000,C 90.000,E1 284.662} C_DIS
LIN {X 0.031,Y -447.390,Z 1337.577,A 0.000,B 0.000,C 90.000,E1 283.883} C_DIS
LIN {X -0.129,Y -451.840,Z 1337.573,A 0.000,B 0.000,C 90.000,E1 283.119} C_DIS
LIN {X 0.189,Y -455.462,Z 1337.568,A 0.000,B 0.000,C 90.000,E1 282.299} C_DIS
LIN {X -0.172,Y -457.475,Z 1337.566,A 0.000,B 0.000,C 90.000,E1 281.827} C_DIS
LIN {X -0.083,Y -459.125,Z 1337.563,A 0.000,B 0.000,C 90.000,E1 281.299} C_DIS
LIN {X -0.068,Y -460.446,Z 1337.560,A 0.000,B 0.000,C 90.000,E1 280.782} C_DIS
LIN {X 0.043,Y -461.359,Z 1337.557,A 0.000,B 0.000,C 90.000,E1 280.254} C_DIS
LIN {X 0.161,Y -461.866,Z 1337.554,A 0.000,B 0.000,C 90.000,E1 279.726} C_DIS
LIN {X 0.205,Y -461.875,Z 1337.551,A 0.000,B 0.000,C 90.000,E1 279.208} C_DIS
LIN {X -0.200,Y -461.496,Z 1337.548,A 0.000,B 0.000,C 90.000,E1 278.746} C_DIS
LIN {X -0.080,Y -460.600,Z 1337.546,A 0.000,B 0.000,C 90.000,E1 278.219} C_DIS
LIN {X -0.030,Y -459.206,Z 1337.543,A 0.000,B 0.000,C 90.000,E1 277.701} C_DIS
LIN {X 0.016,Y -457.301,Z 1337.540,A 0.000,B 0.000,C 90.000,E1 277.182} C_DIS
LIN {X 0.054,Y -454.836,Z 1337.537,A 0.000,B 0.000,C 90.000,E1 276.663} C_DIS
LIN {X 0.076,Y -451.791,Z 1337.534,A 0.000,B 0.000,C 90.000,E1 276.144} C_DIS
LIN {X 0.081,Y -448.139,Z 1337.531,A 0.000,B 0.000,C 90.000,E1 275.625} C_DIS
LIN {X 0.066,Y -443.752,Z 1337.528,A 0.000,B 0.000,C 90.000,E1 275.106} C_DIS
LIN {X 0.026,Y -438.339,Z 1337.526,A 0.000,B 0.000,C 90.000,E1 274.588} C_DIS
LIN {X -0.171,Y -432.295,Z 1337.523,A 0.000,B 0.000,C 90.000,E1 274.131} C_DIS
LIN {X 0.103,Y -426.101,Z 1337.521,A 0.000,B 0.000,C 90.000,E1 273.669} C_DIS
LIN {X -0.153,Y -419.560,Z 1337.518,A 0.000,B 0.000,C 90.000,E1 273.326} C_DIS
LIN {X -0.020,Y -413.089,Z 1337.516,A 0.000,B 0.000,C 90.000,E1 272.980} C_DIS
LIN {X -0.097,Y -406.371,Z 1337.515,A 0.000,B 0.000,C 90.000,E1 272.694} C_DIS
LIN {X 0.084,Y -399.338,Z 1337.513,A 0.000,B 0.000,C 90.000,E1 272.407} C_DIS
LIN {X -0.065,Y -388.600,Z 1337.512,A 0.000,B 0.000,C 90.000,E1 272.121} C_DIS
LIN {X 0.004,Y -381.352,Z 1337.511,A 0.000,B 0.000,C 90.000,E1 271.949} C_DIS
LIN {X -0.117,Y -373.494,Z 1337.510,A 0.000,B 0.000,C 90.000,E1 271.835} C_DIS
LIN {X -0.054,Y -364.338,Z 1337.510,A 0.000,B 0.000,C 90.000,E1 271.718} C_DIS
LIN {X 0.134,Y -351.702,Z 1337.509,A 0.000,B 0.000,C 90.000,E1 271.604} C_DIS
LIN {X 0.076,Y -347.302,Z 1337.509,A 0.000,B 0.000,C 90.000,E1 271.604} C_DIS
LIN {X 0.011,Y -181.330,Z 1337.509,A 0.000,B 0.000,C 90.000,E1 271.604} C_DIS
LIN {X 0.056,Y -181.570,Z 1337.500,A 0.000,B 0.000,C 90.000,E1 270.057} C_DIS
LIN {X 0.013,Y -180.906,Z 1337.474,A 0.000,B 0.000,C 90.000,E1 265.355} C_DIS
LIN {X 0.087,Y -180.684,Z 1337.469,A 0.000,B 0.000,C 90.000,E1 264.489} C_DIS
LIN {X -0.014,Y -178.767,Z 1337.441,A 0.000,B 0.000,C 90.000,E1 259.454} C_DIS
LIN {X 0.057,Y -175.813,Z 1337.413,A 0.000,B 0.000,C 90.000,E1 254.338} C_DIS
LIN {X 0.051,Y -172.000,Z 1337.385,A 0.000,B 0.000,C 90.000,E1 249.209} C_DIS
LIN {X 0.025,Y -171.415,Z 1337.380,A 0.000,B 0.000,C 90.000,E1 248.358} C_DIS
LIN {X 0.073,Y -167.654,Z 1337.356,A 0.000,B 0.000,C 90.000,E1 244.024} C_DIS
LIN {X 0.087,Y -166.321,Z 1337.346,A 0.000,B 0.000,C 90.000,E1 242.281} C_DIS
LIN {X -0.004,Y -163.061,Z 1337.327,A 0.000,B 0.000,C 90.000,E1 238.820} C_DIS
LIN {X 0.041,Y -160.998,Z 1337.312,A 0.000,B 0.000,C 90.000,E1 236.167} C_DIS
LIN {X 0.019,Y -157.744,Z 1337.292,A 0.000,B 0.000,C 90.000,E1 232.637} C_DIS
LIN {X -0.043,Y -155.783,Z 1337.278,A 0.000,B 0.000,C 90.000,E1 229.989} C_DIS
LIN {X 0.012,Y -152.036,Z 1337.253,A 0.000,B 0.000,C 90.000,E1 225.486} C_DIS
LIN {X 0.030,Y -150.285,Z 1337.238,A 0.000,B 0.000,C 90.000,E1 222.771} C_DIS
LIN {X -0.043,Y -147.034,Z 1337.212,A 0.000,B 0.000,C 90.000,E1 218.257} C_DIS
LIN {X -0.051,Y -145.615,Z 1337.197,A 0.000,B 0.000,C 90.000,E1 215.518} C_DIS
LIN {X -0.052,Y -142.999,Z 1337.172,A 0.000,B 0.000,C 90.000,E1 210.924} C_DIS
LIN {X 0.006,Y -141.626,Z 1337.151,A 0.000,B 0.000,C 90.000,E1 207.206} C_DIS
LIN {X -0.069,Y -139.433,Z 1337.115,A 0.000,B 0.000,C 90.000,E1 200.737} C_DIS
LIN {X -0.015,Y -139.164,Z 1337.105,A 0.000,B 0.000,C 90.000,E1 198.852} C_DIS
LIN {X 0.022,Y -138.340,Z 1337.058,A 0.000,B 0.000,C 90.000,E1 190.433} C_DIS
LIN {X 0.030,Y -139.477,Z 1337.006,A 0.000,B 0.000,C 90.000,E1 181.088} C_DIS
LIN {X -0.029,Y -141.060,Z 1336.975,A 0.000,B 0.000,C 90.000,E1 175.527} C_DIS
LIN {X 0.066,Y -142.433,Z 1336.960,A 0.000,B 0.000,C 90.000,E1 172.704} C_DIS
LIN {X -0.014,Y -144.671,Z 1336.934,A 0.000,B 0.000,C 90.000,E1 168.117} C_DIS
LIN {X -0.031,Y -147.257,Z 1336.914,A 0.000,B 0.000,C 90.000,E1 164.448} C_DIS
LIN {X -0.014,Y -150.575,Z 1336.888,A 0.000,B 0.000,C 90.000,E1 159.880} C_DIS
LIN {X 0.065,Y -154.045,Z 1336.868,A 0.000,B 0.000,C 90.000,E1 156.230} C_DIS
LIN {X -0.008,Y -157.462,Z 1336.848,A 0.000,B 0.000,C 90.000,E1 152.666} C_DIS
LIN {X -0.060,Y -161.682,Z 1336.828,A 0.000,B 0.000,C 90.000,E1 149.125} C_DIS
LIN {X -0.043,Y -165.877,Z 1336.809,A 0.000,B 0.000,C 90.000,E1 145.595} C_DIS
LIN {X -0.052,Y -170.856,Z 1336.789,A 0.000,B 0.000,C 90.000,E1 142.110} C_DIS
LIN {X -0.006,Y -175.725,Z 1336.770,A 0.000,B 0.000,C 90.000,E1 138.647} C_DIS
LIN {X -0.015,Y -181.337,Z 1336.751,A 0.000,B 0.000,C 90.000,E1 135.243} C_DIS
LIN {X -0.020,Y -186.825,Z 1336.733,A 0.000,B 0.000,C 90.000,E1 131.881} C_DIS
LIN {X 0.073,Y -191.413,Z 1336.719,A 0.000,B 0.000,C 90.000,E1 129.358} C_DIS
LIN {X 0.006,Y -197.261,Z 1336.701,A 0.000,B 0.000,C 90.000,E1 126.091} C_DIS
LIN {X 0.058,Y -199.190,Z 1336.695,A 0.000,B 0.000,C 90.000,E1 125.105} C_DIS
LIN {X 0.040,Y -309.078,Z 1336.695,A 0.000,B 0.000,C 90.000,E1 125.105} C_DIS
LIN {X -0.109,Y -310.735,Z 1336.695,A 0.000,B 0.000,C 90.000,E1 125.105} C_DIS
LIN {X 0.019,Y -316.598,Z 1336.693,A 0.000,B 0.000,C 90.000,E1 124.771} C_DIS
LIN {X -0.112,Y -319.597,Z 1336.692,A 0.000,B 0.000,C 90.000,E1 124.485} C_DIS
LIN {X -0.115,Y -321.605,Z 1336.690,A 0.000,B 0.000,C 90.000,E1 124.199} C_DIS
LIN {X -0.119,Y -323.175,Z 1336.688,A 0.000,B 0.000,C 90.000,E1 123.913} C_DIS
LIN {X -0.033,Y -324.552,Z 1336.687,A 0.000,B 0.000,C 90.000,E1 123.579} C_DIS
LIN {X 0.055,Y -336.111,Z 1336.669,A 0.000,B 0.000,C 90.000,E1 120.413} C_DIS
LIN {X 0.004,Y -347.898,Z 1336.654,A 0.000,B 0.000,C 90.000,E1 117.641} C_DIS
LIN {X 0.115,Y -361.128,Z 1336.638,A 0.000,B 0.000,C 90.000,E1 114.899} C_DIS
LIN {X 0.207,Y -374.196,Z 1336.625,A 0.000,B 0.000,C 90.000,E1 112.514} C_DIS
LIN {X -0.155,Y -388.586,Z 1336.612,A 0.000,B 0.000,C 90.000,E1 110.248} C_DIS
LIN {X 0.075,Y -404.399,Z 1336.600,A 0.000,B 0.000,C 90.000,E1 107.946} C_DIS
LIN {X 0.077,Y -421.748,Z 1336.587,A 0.000,B 0.000,C 90.000,E1 105.733} C_DIS
LIN {X -0.013,Y -440.737,Z 1336.575,A 0.000,B 0.000,C 90.000,E1 103.592} C_DIS
LIN {X -0.191,Y -460.771,Z 1336.564,A 0.000,B 0.000,C 90.000,E1 101.591} C_DIS
LIN {X 0.221,Y -478.763,Z 1336.555,A 0.000,B 0.000,C 90.000,E1 99.905} C_DIS
LIN {X -0.143,Y -481.014,Z 1336.554,A 0.000,B 0.000,C 90.000,E1 99.726} C_DIS
LIN {X -0.116,Y -482.716,Z 1336.553,A 0.000,B 0.000,C 90.000,E1 99.500} C_DIS
LIN {X -0.234,Y -484.168,Z 1336.551,A 0.000,B 0.000,C 90.000,E1 99.265} C_DIS
LIN {X 0.126,Y -485.249,Z 1336.550,A 0.000,B 0.000,C 90.000,E1 98.973} C_DIS
LIN {X -0.170,Y -486.509,Z 1336.547,A 0.000,B 0.000,C 90.000,E1 98.511} C_DIS
LIN {X 0.023,Y -486.747,Z 1336.544,A 0.000,B 0.000,C 90.000,E1 97.992} C_DIS
LIN {X -0.257,Y -486.001,Z 1336.542,A 0.000,B 0.000,C 90.000,E1 97.530} C_DIS
LIN {X 0.007,Y -484.148,Z 1336.539,A 0.000,B 0.000,C 90.000,E1 97.004} C_DIS
LIN {X -0.164,Y -482.696,Z 1336.538,A 0.000,B 0.000,C 90.000,E1 96.777} C_DIS
LIN {X -0.018,Y -468.422,Z 1336.526,A 0.000,B 0.000,C 90.000,E1 94.759} C_DIS
LIN {X -0.039,Y -456.678,Z 1336.516,A 0.000,B 0.000,C 90.000,E1 92.980} C_DIS
LIN {X 0.070,Y -441.869,Z 1336.504,A 0.000,B 0.000,C 90.000,E1 90.630} C_DIS
LIN {X 0.094,Y -425.483,Z 1336.487,A 0.000,B 0.000,C 90.000,E1 87.707} C_DIS
LIN {X 0.093,Y -415.374,Z 1336.477,A 0.000,B 0.000,C 90.000,E1 85.812} C_DIS
LIN {X -0.180,Y -406.556,Z 1336.468,A 0.000,B 0.000,C 90.000,E1 84.204} C_DIS
LIN {X -0.117,Y -397.611,Z 1336.458,A 0.000,B 0.000,C 90.000,E1 82.527} C_DIS
LIN {X 0.175,Y -388.394,Z 1336.449,A 0.000,B 0.000,C 90.000,E1 80.792} C_DIS
LIN {X -0.027,Y -378.965,Z 1336.439,A 0.000,B 0.000,C 90.000,E1 79.106} C_DIS
LIN {X 0.043,Y -369.312,Z 1336.430,A 0.000,B 0.000,C 90.000,E1 77.353} C_DIS
LIN {X 0.067,Y -357.793,Z 1336.418,A 0.000,B 0.000,C 90.000,E1 75.283} C_DIS
LIN {X -0.078,Y -347.958,Z 1336.408,A 0.000,B 0.000,C 90.000,E1 73.504} C_DIS
LIN {X 0.121,Y -336.307,Z 1336.396,A 0.000,B 0.000,C 90.000,E1 71.329} C_DIS
LIN {X 0.025,Y -323.219,Z 1336.383,A 0.000,B 0.000,C 90.000,E1 68.847} C_DIS
LIN {X -0.170,Y -306.121,Z 1336.363,A 0.000,B 0.000,C 90.000,E1 65.357} C_DIS
LIN {X 0.132,Y -296.246,Z 1336.350,A 0.000,B 0.000,C 90.000,E1 62.999} C_DIS
LIN {X 0.091,Y -287.499,Z 1336.337,A 0.000,B 0.000,C 90.000,E1 60.667} C_DIS
LIN {X -0.133,Y -278.752,Z 1336.322,A 0.000,B 0.000,C 90.000,E1 57.995} C_DIS
LIN {X 0.147,Y -268.950,Z 1336.303,A 0.000,B 0.000,C 90.000,E1 54.482} C_DIS
LIN {X 0.030,Y -261.620,Z 1336.287,A 0.000,B 0.000,C 90.000,E1 51.698} C_DIS
LIN {X -0.107,Y -252.976,Z 1336.267,A 0.000,B 0.000,C 90.000,E1 48.162} C_DIS
LIN {X -0.012,Y -246.408,Z 1336.251,A 0.000,B 0.000,C 90.000,E1 45.243} C_DIS
LIN {X 0.054,Y -238.667,Z 1336.231,A 0.000,B 0.000,C 90.000,E1 41.553} C_DIS
LIN {X 0.099,Y -231.682,Z 1336.210,A 0.000,B 0.000,C 90.000,E1 37.810} C_DIS
LIN {X 0.042,Y -225.586,Z 1336.189,A 0.000,B 0.000,C 90.000,E1 34.040} C_DIS
LIN {X 0.048,Y -220.493,Z 1336.168,A 0.000,B 0.000,C 90.000,E1 30.207} C_DIS
LIN {X -0.075,Y -215.717,Z 1336.142,A 0.000,B 0.000,C 90.000,E1 25.591} C_DIS
LIN {X 0.053,Y -211.923,Z 1336.116,A 0.000,B 0.000,C 90.000,E1 20.865} C_DIS
LIN {X 0.097,Y -209.155,Z 1336.094,A 0.000,B 0.000,C 90.000,E1 16.913} C_DIS
LIN {X -0.108,Y -206.574,Z 1336.072,A 0.000,B 0.000,C 90.000,E1 13.008} C_DIS
LIN {X -0.090,Y -203.735,Z 1336.046,A 0.000,B 0.000,C 90.000,E1 8.219} C_DIS
LIN {X -0.006,Y -201.933,Z 1336.023,A 0.000,B 0.000,C 90.000,E1 4.188} C_DIS
LIN {X -0.080,Y -200.290,Z 1335.984,A 0.000,B 0.000,C 90.000,E1 357.135} C_DIS
LIN {X -0.024,Y -201.053,Z 1335.939,A 0.000,B 0.000,C 90.000,E1 349.050} C_DIS
LIN {X 0.036,Y -203.928,Z 1335.903,A 0.000,B 0.000,C 90.000,E1 342.598} C_DIS
LIN {X 0.070,Y -207.570,Z 1335.877,A 0.000,B 0.000,C 90.000,E1 337.794} C_DIS
LIN {X 0.016,Y -211.747,Z 1335.855,A 0.000,B 0.000,C 90.000,E1 333.845} C_DIS
LIN {X 0.003,Y -216.874,Z 1335.833,A 0.000,B 0.000,C 90.000,E1 329.921} C_DIS
LIN {X 0.121,Y -223.116,Z 1335.811,A 0.000,B 0.000,C 90.000,E1 326.008} C_DIS
LIN {X 0.072,Y -230.385,Z 1335.790,A 0.000,B 0.000,C 90.000,E1 322.190} C_DIS
LIN {X -0.044,Y -238.852,Z 1335.769,A 0.000,B 0.000,C 90.000,E1 318.447} C_DIS
LIN {X 0.079,Y -247.424,Z 1335.751,A 0.000,B 0.000,C 90.000,E1 315.081} C_DIS
LIN {X -0.103,Y -253.804,Z 1335.738,A 0.000,B 0.000,C 90.000,E1 312.933} C_DIS
LIN {X 0.112,Y -263.474,Z 1335.722,A 0.000,B 0.000,C 90.000,E1 310.011} C_DIS
LIN {X 0.121,Y -271.641,Z 1335.711,A 0.000,B 0.000,C 90.000,E1 307.890} C_DIS
LIN {X 0.065,Y -282.293,Z 1335.697,A 0.000,B 0.000,C 90.000,E1 305.471} C_DIS
LIN {X -0.060,Y -292.542,Z 1335.686,A 0.000,B 0.000,C 90.000,E1 303.452} C_DIS
LIN {X 0.086,Y -302.041,Z 1335.677,A 0.000,B 0.000,C 90.000,E1 301.750} C_DIS
LIN {X -0.043,Y -312.614,Z 1335.667,A 0.000,B 0.000,C 90.000,E1 300.129} C_DIS
LIN {X 0.041,Y -326.869,Z 1335.657,A 0.000,B 0.000,C 90.000,E1 298.180} C_DIS
LIN {X -0.105,Y -347.829,Z 1335.643,A 0.000,B 0.000,C 90.000,E1 295.720} C_DIS
LIN {X 0.004,Y -361.025,Z 1335.635,A 0.000,B 0.000,C 90.000,E1 294.207} C_DIS
LIN {X -0.138,Y -373.912,Z 1335.626,A 0.000,B 0.000,C 90.000,E1 292.770} C_DIS
LIN {X 0.065,Y -383.848,Z 1335.620,A 0.000,B 0.000,C 90.000,E1 291.589} C_DIS
LIN {X -0.031,Y -398.494,Z 1335.610,A 0.000,B 0.000,C 90.000,E1 289.885} C_DIS
LIN {X 0.146,Y -413.285,Z 1335.601,A 0.000,B 0.000,C 90.000,E1 288.181} C_DIS
LIN {X 0.062,Y -422.963,Z 1335.595,A 0.000,B 0.000,C 90.000,E1 287.094} C_DIS
LIN {X -0.034,Y -432.088,Z 1335.589,A 0.000,B 0.000,C 90.000,E1 286.024} C_DIS
LIN {X 0.210,Y -438.380,Z 1335.585,A 0.000,B 0.000,C 90.000,E1 285.190} C_DIS
LIN {X -0.031,Y -444.024,Z 1335.580,A 0.000,B 0.000,C 90.000,E1 284.426} C_DIS
LIN {X 0.090,Y -447.433,Z 1335.577,A 0.000,B 0.000,C 90.000,E1 283.883} C_DIS
LIN {X -0.070,Y -451.874,Z 1335.573,A 0.000,B 0.000,C 90.000,E1 283.119} C_DIS
LIN {X -0.196,Y -455.524,Z 1335.568,A 0.000,B 0.000,C 90.000,E1 282.355} C_DIS
LIN {X -0.111,Y -457.569,Z 1335.566,A 0.000,B 0.000,C 90.000,E1 281.827} C_DIS
LIN {X -0.015,Y -459.220,Z 1335.563,A 0.000,B 0.000,C 90.000,E1 281.299} C_DIS
LIN {X 0.000,Y -460.536,Z 1335.560,A 0.000,B 0.000,C 90.000,E1 280.782} C_DIS
LIN {X 0.113,Y -461.503,Z 1335.557,A 0.000,B 0.000,C 90.000,E1 280.254} C_DIS
LIN {X 0.230,Y -462.033,Z 1335.554,A 0.000,B 0.000,C 90.000,E1 279.726} C_DIS
LIN {X -0.180,Y -462.136,Z 1335.551,A 0.000,B 0.000,C 90.000,E1 279.265} C_DIS
LIN {X -0.128,Y -461.727,Z 1335.548,A 0.000,B 0.000,C 90.000,E1 278.746} C_DIS
LIN {X -0.007,Y -460.877,Z 1335.546,A 0.000,B 0.000,C 90.000,E1 278.219} C_DIS
LIN {X 0.044,Y -459.571,Z 1335.543,A 0.000,B 0.000,C 90.000,E1 277.701} C_DIS
LIN {X 0.091,Y -457.703,Z 1335.540,A 0.000,B 0.000,C 90.000,E1 277.182} C_DIS
LIN {X 0.132,Y -455.295,Z 1335.537,A 0.000,B 0.000,C 90.000,E1 276.663} C_DIS
LIN {X 0.155,Y -452.272,Z 1335.534,A 0.000,B 0.000,C 90.000,E1 276.144} C_DIS
LIN {X 0.162,Y -448.720,Z 1335.531,A 0.000,B 0.000,C 90.000,E1 275.625} C_DIS
LIN {X 0.149,Y -444.390,Z 1335.528,A 0.000,B 0.000,C 90.000,E1 275.106} C_DIS
LIN {X 0.112,Y -439.113,Z 1335.526,A 0.000,B 0.000,C 90.000,E1 274.588} C_DIS
LIN {X -0.144,Y -433.098,Z 1335.523,A 0.000,B 0.000,C 90.000,E1 274.131} C_DIS
LIN {X 0.090,Y -426.863,Z 1335.521,A 0.000,B 0.000,C 90.000,E1 273.669} C_DIS
LIN {X -0.143,Y -420.556,Z 1335.518,A 0.000,B 0.000,C 90.000,E1 273.326} C_DIS
LIN {X -0.033,Y -414.145,Z 1335.516,A 0.000,B 0.000,C 90.000,E1 272.980} C_DIS
LIN {X -0.156,Y -407.404,Z 1335.515,A 0.000,B 0.000,C 90.000,E1 272.694} C_DIS
LIN {X -0.029,Y -400.279,Z 1335.513,A 0.000,B 0.000,C 90.000,E1 272.407} C_DIS
LIN {X 0.001,Y -392.818,Z 1335.512,A 0.000,B 0.000,C 90.000,E1 272.178} C_DIS
LIN {X -0.063,Y -385.444,Z 1335.511,A 0.000,B 0.000,C 90.000,E1 272.007} C_DIS
LIN {X 0.086,Y -377.734,Z 1335.510,A 0.000,B 0.000,C 90.000,E1 271.835} C_DIS
LIN {X 0.057,Y -369.166,Z 1335.510,A 0.000,B 0.000,C 90.000,E1 271.718} C_DIS
LIN {X 0.071,Y -355.451,Z 1335.509,A 0.000,B 0.000,C 90.000,E1 271.604} C_DIS
LIN {X -0.097,Y -346.350,Z 1335.509,A 0.000,B 0.000,C 90.000,E1 271.604} C_DIS
LIN {X -0.079,Y -181.336,Z 1335.509,A 0.000,B 0.000,C 90.000,E1 271.604} C_DIS
LIN {X -0.033,Y -181.567,Z 1335.500,A 0.000,B 0.000,C 90.000,E1 270.057} C_DIS
LIN {X -0.076,Y -180.905,Z 1335.474,A 0.000,B 0.000,C 90.000,E1 265.355} C_DIS
LIN {X -0.002,Y -180.669,Z 1335.469,A 0.000,B 0.000,C 90.000,E1 264.489} C_DIS
LIN {X 0.073,Y -178.751,Z 1335.441,A 0.000,B 0.000,C 90.000,E1 259.398} C_DIS
LIN {X -0.030,Y -175.797,Z 1335.413,A 0.000,B 0.000,C 90.000,E1 254.338} C_DIS
LIN {X -0.036,Y -171.983,Z 1335.384,A 0.000,B 0.000,C 90.000,E1 249.209} C_DIS
LIN {X 0.003,Y -171.389,Z 1335.380,A 0.000,B 0.000,C 90.000,E1 248.337} C_DIS
LIN {X -0.012,Y -167.632,Z 1335.356,A 0.000,B 0.000,C 90.000,E1 244.024} C_DIS
LIN {X 0.003,Y -166.289,Z 1335.346,A 0.000,B 0.000,C 90.000,E1 242.281} C_DIS
LIN {X -0.003,Y -163.037,Z 1335.327,A 0.000,B 0.000,C 90.000,E1 238.791} C_DIS
LIN {X -0.040,Y -160.967,Z 1335.312,A 0.000,B 0.000,C 90.000,E1 236.167} C_DIS
LIN {X -0.063,Y -157.719,Z 1335.292,A 0.000,B 0.000,C 90.000,E1 232.637} C_DIS
LIN {X 0.095,Y -155.759,Z 1335.277,A 0.000,B 0.000,C 90.000,E1 229.908} C_DIS
LIN {X -0.067,Y -152.015,Z 1335.253,A 0.000,B 0.000,C 90.000,E1 225.486} C_DIS
LIN {X -0.049,Y -150.262,Z 1335.238,A 0.000,B 0.000,C 90.000,E1 222.771} C_DIS
LIN {X -0.031,Y -147.016,Z 1335.212,A 0.000,B 0.000,C 90.000,E1 218.222} C_DIS
LIN {X -0.011,Y -145.599,Z 1335.197,A 0.000,B 0.000,C 90.000,E1 215.471} C_DIS
LIN {X -0.006,Y -142.985,Z 1335.172,A 0.000,B 0.000,C 90.000,E1 210.875} C_DIS
LIN {X -0.006,Y -141.612,Z 1335.151,A 0.000,B 0.000,C 90.000,E1 207.180} C_DIS
LIN {X 0.035,Y -139.428,Z 1335.115,A 0.000,B 0.000,C 90.000,E1 200.663} C_DIS
LIN {X -0.046,Y -139.157,Z 1335.104,A 0.000,B 0.000,C 90.000,E1 198.833} C_DIS
LIN {X -0.028,Y -138.343,Z 1335.058,A 0.000,B 0.000,C 90.000,E1 190.423} C_DIS
LIN {X -0.046,Y -139.481,Z 1335.006,A 0.000,B 0.000,C 90.000,E1 181.088} C_DIS
LIN {X 0.034,Y -141.073,Z 1334.975,A 0.000,B 0.000,C 90.000,E1 175.469} C_DIS
LIN {X -0.012,Y -142.449,Z 1334.959,A 0.000,B 0.000,C 90.000,E1 172.704} C_DIS
LIN {X 0.078,Y -144.690,Z 1334.934,A 0.000,B 0.000,C 90.000,E1 168.049} C_DIS
LIN {X 0.031,Y -147.282,Z 1334.913,A 0.000,B 0.000,C 90.000,E1 164.393} C_DIS
LIN {X 0.048,Y -150.600,Z 1334.888,A 0.000,B 0.000,C 90.000,E1 159.826} C_DIS
LIN {X -0.016,Y -154.074,Z 1334.868,A 0.000,B 0.000,C 90.000,E1 156.230} C_DIS
LIN {X 0.049,Y -157.494,Z 1334.848,A 0.000,B 0.000,C 90.000,E1 152.615} C_DIS
LIN {X -0.005,Y -161.722,Z 1334.828,A 0.000,B 0.000,C 90.000,E1 149.076} C_DIS
LIN {X 0.009,Y -165.915,Z 1334.809,A 0.000,B 0.000,C 90.000,E1 145.548} C_DIS
LIN {X -0.004,Y -170.901,Z 1334.789,A 0.000,B 0.000,C 90.000,E1 142.065} C_DIS
LIN {X 0.023,Y -175.769,Z 1334.770,A 0.000,B 0.000,C 90.000,E1 138.609} C_DIS
LIN {X 0.024,Y -181.378,Z 1334.751,A 0.000,B 0.000,C 90.000,E1 135.202} C_DIS
LIN {X 0.027,Y -186.874,Z 1334.732,A 0.000,B 0.000,C 90.000,E1 131.838} C_DIS
LIN {X -0.020,Y -191.457,Z 1334.719,A 0.000,B 0.000,C 90.000,E1 129.358} C_DIS
LIN {X -0.088,Y -197.313,Z 1334.700,A 0.000,B 0.000,C 90.000,E1 126.091} C_DIS
LIN {X 0.032,Y -199.206,Z 1334.695,A 0.000,B 0.000,C 90.000,E1 125.105} C_DIS
LIN {X 0.014,Y -309.190,Z 1334.695,A 0.000,B 0.000,C 90.000,E1 125.105} C_DIS
LIN {X 0.177,Y -311.561,Z 1334.695,A 0.000,B 0.000,C 90.000,E1 125.025} C_DIS
LIN {X 0.049,Y -316.864,Z 1334.693,A 0.000,B 0.000,C 90.000,E1 124.739} C_DIS
LIN {X -0.083,Y -319.774,Z 1334.691,A 0.000,B 0.000,C 90.000,E1 124.452} C_DIS
LIN {X 0.143,Y -321.778,Z 1334.690,A 0.000,B 0.000,C 90.000,E1 124.119} C_DIS
LIN {X -0.076,Y -323.342,Z 1334.688,A 0.000,B 0.000,C 90.000,E1 123.865} C_DIS
LIN {X 0.191,Y -324.682,Z 1334.686,A 0.000,B 0.000,C 90.000,E1 123.499} C_DIS
LIN {X -0.005,Y -336.245,Z 1334.669,A 0.000,B 0.000,C 90.000,E1 120.384} C_DIS
LIN {X 0.078,Y -348.052,Z 1334.653,A 0.000,B 0.000,C 90.000,E1 117.590} C_DIS
LIN {X -0.124,Y -361.302,Z 1334.638,A 0.000,B 0.000,C 90.000,E1 114.899} C_DIS
LIN {X -0.036,Y -374.389,Z 1334.625,A 0.000,B 0.000,C 90.000,E1 112.514} C_DIS
LIN {X 0.096,Y -388.801,Z 1334.612,A 0.000,B 0.000,C 90.000,E1 110.174} C_DIS
LIN {X -0.177,Y -404.638,Z 1334.600,A 0.000,B 0.000,C 90.000,E1 107.946} C_DIS
LIN {X -0.066,Y -422.012,Z 1334.587,A 0.000,B 0.000,C 90.000,E1 105.717} C_DIS
LIN {X 0.156,Y -441.026,Z 1334.575,A 0.000,B 0.000,C 90.000,E1 103.536} C_DIS
LIN {X 0.010,Y -461.070,Z 1334.564,A 0.000,B 0.000,C 90.000,E1 101.535} C_DIS
LIN {X -0.021,Y -479.064,Z 1334.555,A 0.000,B 0.000,C 90.000,E1 99.905} C_DIS
LIN {X 0.061,Y -481.231,Z 1334.554,A 0.000,B 0.000,C 90.000,E1 99.670} C_DIS
LIN {X 0.064,Y -482.873,Z 1334.552,A 0.000,B 0.000,C 90.000,E1 99.443} C_DIS
LIN {X -0.052,Y -484.254,Z 1334.551,A 0.000,B 0.000,C 90.000,E1 99.208} C_DIS
LIN {X -0.171,Y -485.277,Z 1334.550,A 0.000,B 0.000,C 90.000,E1 98.973} C_DIS
LIN {X 0.013,Y -486.443,Z 1334.547,A 0.000,B 0.000,C 90.000,E1 98.454} C_DIS
LIN {X 0.208,Y -486.596,Z 1334.544,A 0.000,B 0.000,C 90.000,E1 97.936} C_DIS
LIN {X -0.009,Y -485.762,Z 1334.542,A 0.000,B 0.000,C 90.000,E1 97.466} C_DIS
LIN {X 0.190,Y -483.800,Z 1334.539,A 0.000,B 0.000,C 90.000,E1 96.947} C_DIS
LIN {X 0.019,Y -482.274,Z 1334.537,A 0.000,B 0.000,C 90.000,E1 96.720} C_DIS
LIN {X -0.156,Y -469.671,Z 1334.528,A 0.000,B 0.000,C 90.000,E1 94.992} C_DIS
LIN {X -0.145,Y -457.881,Z 1334.518,A 0.000,B 0.000,C 90.000,E1 93.212} C_DIS
LIN {X 0.025,Y -442.985,Z 1334.505,A 0.000,B 0.000,C 90.000,E1 90.859} C_DIS
LIN {X 0.080,Y -426.496,Z 1334.489,A 0.000,B 0.000,C 90.000,E1 87.936} C_DIS
LIN {X 0.078,Y -416.422,Z 1334.478,A 0.000,B 0.000,C 90.000,E1 86.045} C_DIS
LIN {X -0.144,Y -407.609,Z 1334.469,A 0.000,B 0.000,C 90.000,E1 84.432} C_DIS
LIN {X -0.108,Y -398.690,Z 1334.460,A 0.000,B 0.000,C 90.000,E1 82.761} C_DIS
LIN {X -0.186,Y -389.522,Z 1334.450,A 0.000,B 0.000,C 90.000,E1 81.084} C_DIS
LIN {X 0.013,Y -380.118,Z 1334.441,A 0.000,B 0.000,C 90.000,E1 79.342} C_DIS
LIN {X 0.101,Y -370.500,Z 1334.431,A 0.000,B 0.000,C 90.000,E1 77.589} C_DIS
LIN {X 0.142,Y -358.995,Z 1334.420,A 0.000,B 0.000,C 90.000,E1 75.519} C_DIS
LIN {X 0.017,Y -349.155,Z 1334.410,A 0.000,B 0.000,C 90.000,E1 73.740} C_DIS
LIN {X 0.140,Y -337.538,Z 1334.398,A 0.000,B 0.000,C 90.000,E1 71.583} C_DIS
LIN {X 0.139,Y -322.782,Z 1334.382,A 0.000,B 0.000,C 90.000,E1 68.773} C_DIS
LIN {X -0.067,Y -305.728,Z 1334.363,A 0.000,B 0.000,C 90.000,E1 65.281} C_DIS
LIN {X 0.095,Y -295.894,Z 1334.350,A 0.000,B 0.000,C 90.000,E1 62.948} C_DIS
LIN {X 0.183,Y -287.191,Z 1334.337,A 0.000,B 0.000,C 90.000,E1 60.589} C_DIS
LIN {X -0.131,Y -276.461,Z 1334.318,A 0.000,B 0.000,C 90.000,E1 57.248} C_DIS
LIN {X 0.013,Y -266.884,Z 1334.299,A 0.000,B 0.000,C 90.000,E1 53.749} C_DIS
LIN {X -0.047,Y -257.900,Z 1334.279,A 0.000,B 0.000,C 90.000,E1 50.231} C_DIS
LIN {X 0.033,Y -249.544,Z 1334.259,A 0.000,B 0.000,C 90.000,E1 46.620} C_DIS
LIN {X 0.004,Y -241.561,Z 1334.239,A 0.000,B 0.000,C 90.000,E1 42.975} C_DIS
LIN {X -0.047,Y -234.271,Z 1334.218,A 0.000,B 0.000,C 90.000,E1 39.277} C_DIS
LIN {X -0.065,Y -227.803,Z 1334.197,A 0.000,B 0.000,C 90.000,E1 35.518} C_DIS
LIN {X 0.064,Y -222.323,Z 1334.176,A 0.000,B 0.000,C 90.000,E1 31.671} C_DIS
LIN {X 0.018,Y -217.121,Z 1334.150,A 0.000,B 0.000,C 90.000,E1 27.052} C_DIS
LIN {X -0.035,Y -213.047,Z 1334.124,A 0.000,B 0.000,C 90.000,E1 22.386} C_DIS
LIN {X 0.111,Y -210.109,Z 1334.103,A 0.000,B 0.000,C 90.000,E1 18.417} C_DIS
LIN {X -0.053,Y -207.963,Z 1334.085,A 0.000,B 0.000,C 90.000,E1 15.300} C_DIS
LIN {X -0.033,Y -205.912,Z 1334.067,A 0.000,B 0.000,C 90.000,E1 12.119} C_DIS
LIN {X -0.086,Y -202.809,Z 1334.036,A 0.000,B 0.000,C 90.000,E1 6.543} C_DIS
LIN {X -0.085,Y -200.776,Z 1334.005,A 0.000,B 0.000,C 90.000,E1 0.917} C_DIS
LIN {X 0.085,Y -200.121,Z 1333.970,A 0.000,B 0.000,C 90.000,E1 354.666} C_DIS
LIN {X 0.071,Y -201.569,Z 1333.930,A 0.000,B 0.000,C 90.000,E1 347.409} C_DIS
LIN {X -0.049,Y -204.483,Z 1333.899,A 0.000,B 0.000,C 90.000,E1 341.819} C_DIS
LIN {X -0.119,Y -208.417,Z 1333.872,A 0.000,B 0.000,C 90.000,E1 337.050} C_DIS
LIN {X 0.036,Y -212.796,Z 1333.850,A 0.000,B 0.000,C 90.000,E1 333.050} C_DIS
LIN {X 0.066,Y -218.159,Z 1333.829,A 0.000,B 0.000,C 90.000,E1 329.125} C_DIS
LIN {X 0.034,Y -224.629,Z 1333.807,A 0.000,B 0.000,C 90.000,E1 325.261} C_DIS
LIN {X 0.082,Y -230.496,Z 1333.790,A 0.000,B 0.000,C 90.000,E1 322.190} C_DIS
LIN {X -0.029,Y -238.954,Z 1333.769,A 0.000,B 0.000,C 90.000,E1 318.447} C_DIS
LIN {X -0.092,Y -248.526,Z 1333.749,A 0.000,B 0.000,C 90.000,E1 314.757} C_DIS
LIN {X 0.106,Y -255.040,Z 1333.736,A 0.000,B 0.000,C 90.000,E1 312.528} C_DIS
LIN {X -0.017,Y -264.855,Z 1333.720,A 0.000,B 0.000,C 90.000,E1 309.688} C_DIS
LIN {X 0.008,Y -273.194,Z 1333.709,A 0.000,B 0.000,C 90.000,E1 307.569} C_DIS
LIN {X -0.136,Y -282.395,Z 1333.697,A 0.000,B 0.000,C 90.000,E1 305.518} C_DIS
LIN {X -0.028,Y -292.654,Z 1333.686,A 0.000,B 0.000,C 90.000,E1 303.452} C_DIS
LIN {X -0.137,Y -302.147,Z 1333.677,A 0.000,B 0.000,C 90.000,E1 301.799} C_DIS
LIN {X -0.005,Y -312.716,Z 1333.667,A 0.000,B 0.000,C 90.000,E1 300.129} C_DIS
LIN {X 0.082,Y -326.949,Z 1333.657,A 0.000,B 0.000,C 90.000,E1 298.180} C_DIS
LIN {X 0.030,Y -347.724,Z 1333.643,A 0.000,B 0.000,C 90.000,E1 295.720} C_DIS
LIN {X -0.057,Y -360.727,Z 1333.635,A 0.000,B 0.000,C 90.000,E1 294.259} C_DIS
LIN {X 0.064,Y -373.714,Z 1333.627,A 0.000,B 0.000,C 90.000,E1 292.770} C_DIS
LIN {X -0.112,Y -386.108,Z 1333.619,A 0.000,B 0.000,C 90.000,E1 291.354} C_DIS
LIN {X 0.150,Y -403.190,Z 1333.607,A 0.000,B 0.000,C 90.000,E1 289.322} C_DIS
LIN {X 0.050,Y -415.538,Z 1333.600,A 0.000,B 0.000,C 90.000,E1 287.946} C_DIS
LIN {X -0.009,Y -425.169,Z 1333.594,A 0.000,B 0.000,C 90.000,E1 286.858} C_DIS
LIN {X -0.078,Y -434.093,Z 1333.588,A 0.000,B 0.000,C 90.000,E1 285.788} C_DIS
LIN {X 0.178,Y -440.201,Z 1333.583,A 0.000,B 0.000,C 90.000,E1 284.954} C_DIS
LIN {X 0.068,Y -445.650,Z 1333.579,A 0.000,B 0.000,C 90.000,E1 284.175} C_DIS
LIN {X -0.114,Y -450.384,Z 1333.574,A 0.000,B 0.000,C 90.000,E1 283.411} C_DIS
LIN {X 0.193,Y -454.382,Z 1333.570,A 0.000,B 0.000,C 90.000,E1 282.591} C_DIS
LIN {X 0.091,Y -457.576,Z 1333.566,A 0.000,B 0.000,C 90.000,E1 281.827} C_DIS
LIN {X 0.189,Y -459.270,Z 1333.563,A 0.000,B 0.000,C 90.000,E1 281.299} C_DIS
LIN {X -0.249,Y -460.616,Z 1333.560,A 0.000,B 0.000,C 90.000,E1 280.838} C_DIS
LIN {X -0.136,Y -461.600,Z 1333.557,A 0.000,B 0.000,C 90.000,E1 280.310} C_DIS
LIN {X -0.098,Y -462.183,Z 1333.554,A 0.000,B 0.000,C 90.000,E1 279.792} C_DIS
LIN {X 0.026,Y -462.331,Z 1333.552,A 0.000,B 0.000,C 90.000,E1 279.265} C_DIS
LIN {X 0.078,Y -462.000,Z 1333.549,A 0.000,B 0.000,C 90.000,E1 278.746} C_DIS
LIN {X 0.201,Y -461.227,Z 1333.546,A 0.000,B 0.000,C 90.000,E1 278.219} C_DIS
LIN {X -0.203,Y -459.973,Z 1333.543,A 0.000,B 0.000,C 90.000,E1 277.757} C_DIS
LIN {X -0.154,Y -458.171,Z 1333.540,A 0.000,B 0.000,C 90.000,E1 277.239} C_DIS
LIN {X -0.109,Y -455.835,Z 1333.537,A 0.000,B 0.000,C 90.000,E1 276.720} C_DIS
LIN {X -0.083,Y -452.892,Z 1333.534,A 0.000,B 0.000,C 90.000,E1 276.201} C_DIS
LIN {X -0.071,Y -449.403,Z 1333.531,A 0.000,B 0.000,C 90.000,E1 275.682} C_DIS
LIN {X -0.078,Y -445.170,Z 1333.529,A 0.000,B 0.000,C 90.000,E1 275.163} C_DIS
LIN {X -0.109,Y -440.052,Z 1333.526,A 0.000,B 0.000,C 90.000,E1 274.645} C_DIS
LIN {X 0.000,Y -434.098,Z 1333.523,A 0.000,B 0.000,C 90.000,E1 274.131} C_DIS
LIN {X 0.162,Y -427.889,Z 1333.521,A 0.000,B 0.000,C 90.000,E1 273.669} C_DIS
LIN {X -0.168,Y -421.467,Z 1333.518,A 0.000,B 0.000,C 90.000,E1 273.326} C_DIS
LIN {X -0.107,Y -415.000,Z 1333.516,A 0.000,B 0.000,C 90.000,E1 272.980} C_DIS
LIN {X 0.171,Y -408.287,Z 1333.515,A 0.000,B 0.000,C 90.000,E1 272.636} C_DIS
LIN {X -0.113,Y -401.309,Z 1333.513,A 0.000,B 0.000,C 90.000,E1 272.407} C_DIS
LIN {X -0.135,Y -393.744,Z 1333.512,A 0.000,B 0.000,C 90.000,E1 272.178} C_DIS
LIN {X 0.159,Y -386.106,Z 1333.511,A 0.000,B 0.000,C 90.000,E1 271.949} C_DIS
LIN {X -0.079,Y -378.323,Z 1333.510,A 0.000,B 0.000,C 90.000,E1 271.835} C_DIS
LIN {X -0.118,Y -369.714,Z 1333.509,A 0.000,B 0.000,C 90.000,E1 271.718} C_DIS
LIN {X -0.105,Y -355.608,Z 1333.509,A 0.000,B 0.000,C 90.000,E1 271.604} C_DIS
LIN {X 0.135,Y -350.474,Z 1333.509,A 0.000,B 0.000,C 90.000,E1 271.547} C_DIS
LIN {X 0.041,Y -181.339,Z 1333.509,A 0.000,B 0.000,C 90.000,E1 271.547} C_DIS
LIN {X 0.060,Y -181.563,Z 1333.500,A 0.000,B 0.000,C 90.000,E1 270.000} C_DIS
LIN {X 0.016,Y -180.903,Z 1333.474,A 0.000,B 0.000,C 90.000,E1 265.298} C_DIS
LIN {X -0.034,Y -180.246,Z 1333.465,A 0.000,B 0.000,C 90.000,E1 263.628} C_DIS
LIN {X -0.016,Y -178.734,Z 1333.441,A 0.000,B 0.000,C 90.000,E1 259.398} C_DIS
LIN {X 0.051,Y -175.781,Z 1333.413,A 0.000,B 0.000,C 90.000,E1 254.283} C_DIS
LIN {X 0.039,Y -171.966,Z 1333.384,A 0.000,B 0.000,C 90.000,E1 249.156} C_DIS
LIN {X 0.077,Y -171.363,Z 1333.380,A 0.000,B 0.000,C 90.000,E1 248.284} C_DIS
LIN {X 0.054,Y -167.611,Z 1333.355,A 0.000,B 0.000,C 90.000,E1 243.973} C_DIS
LIN {X 0.066,Y -166.259,Z 1333.346,A 0.000,B 0.000,C 90.000,E1 242.231} C_DIS
LIN {X 0.053,Y -163.013,Z 1333.326,A 0.000,B 0.000,C 90.000,E1 238.742} C_DIS
LIN {X -0.034,Y -160.937,Z 1333.312,A 0.000,B 0.000,C 90.000,E1 236.135} C_DIS
LIN {X 0.076,Y -157.696,Z 1333.292,A 0.000,B 0.000,C 90.000,E1 232.557} C_DIS
LIN {X 0.015,Y -155.735,Z 1333.277,A 0.000,B 0.000,C 90.000,E1 229.908} C_DIS
LIN {X 0.068,Y -151.994,Z 1333.252,A 0.000,B 0.000,C 90.000,E1 225.405} C_DIS
LIN {X 0.084,Y -150.239,Z 1333.237,A 0.000,B 0.000,C 90.000,E1 222.690} C_DIS
LIN {X 0.006,Y -146.998,Z 1333.212,A 0.000,B 0.000,C 90.000,E1 218.177} C_DIS
LIN {X -0.003,Y -145.583,Z 1333.197,A 0.000,B 0.000,C 90.000,E1 215.438} C_DIS
LIN {X -0.009,Y -142.972,Z 1333.171,A 0.000,B 0.000,C 90.000,E1 210.846} C_DIS
LIN {X 0.043,Y -141.598,Z 1333.151,A 0.000,B 0.000,C 90.000,E1 207.129} C_DIS
LIN {X -0.040,Y -139.423,Z 1333.115,A 0.000,B 0.000,C 90.000,E1 200.663} C_DIS
LIN {X 0.010,Y -139.150,Z 1333.104,A 0.000,B 0.000,C 90.000,E1 198.779} C_DIS
LIN {X 0.033,Y -138.345,Z 1333.058,A 0.000,B 0.000,C 90.000,E1 190.366} C_DIS
LIN {X 0.018,Y -139.486,Z 1333.006,A 0.000,B 0.000,C 90.000,E1 181.031} C_DIS
LIN {X -0.042,Y -141.086,Z 1332.975,A 0.000,B 0.000,C 90.000,E1 175.469} C_DIS
LIN {X 0.053,Y -142.464,Z 1332.959,A 0.000,B 0.000,C 90.000,E1 172.648} C_DIS
LIN {X 0.002,Y -144.708,Z 1332.934,A 0.000,B 0.000,C 90.000,E1 168.049} C_DIS
LIN {X -0.047,Y -147.306,Z 1332.913,A 0.000,B 0.000,C 90.000,E1 164.393} C_DIS
LIN {X -0.032,Y -150.626,Z 1332.888,A 0.000,B 0.000,C 90.000,E1 159.826} C_DIS
LIN {X 0.044,Y -154.102,Z 1332.868,A 0.000,B 0.000,C 90.000,E1 156.177} C_DIS
LIN {X -0.032,Y -157.526,Z 1332.848,A 0.000,B 0.000,C 90.000,E1 152.615} C_DIS
LIN {X -0.088,Y -161.760,Z 1332.828,A 0.000,B 0.000,C 90.000,E1 149.076} C_DIS
LIN {X 0.018,Y -165.953,Z 1332.808,A 0.000,B 0.000,C 90.000,E1 145.515} C_DIS
LIN {X 0.015,Y -170.945,Z 1332.789,A 0.000,B 0.000,C 90.000,E1 142.029} C_DIS
LIN {X -0.065,Y -175.813,Z 1332.770,A 0.000,B 0.000,C 90.000,E1 138.609} C_DIS
LIN {X 0.062,Y -181.420,Z 1332.751,A 0.000,B 0.000,C 90.000,E1 135.162} C_DIS
LIN {X -0.063,Y -186.923,Z 1332.732,A 0.000,B 0.000,C 90.000,E1 131.838} C_DIS
LIN {X 0.010,Y -191.503,Z 1332.719,A 0.000,B 0.000,C 90.000,E1 129.322} C_DIS
LIN {X 0.095,Y -197.367,Z 1332.700,A 0.000,B 0.000,C 90.000,E1 126.011} C_DIS
LIN {X 0.026,Y -199.209,Z 1332.695,A 0.000,B 0.000,C 90.000,E1 125.105} C_DIS
LIN {X -0.010,Y -309.279,Z 1332.695,A 0.000,B 0.000,C 90.000,E1 125.105} C_DIS
LIN {X 0.135,Y -314.418,Z 1332.694,A 0.000,B 0.000,C 90.000,E1 124.898} C_DIS
LIN {X 0.074,Y -316.764,Z 1332.693,A 0.000,B 0.000,C 90.000,E1 124.739} C_DIS
LIN {X 0.031,Y -319.947,Z 1332.691,A 0.000,B 0.000,C 90.000,E1 124.405} C_DIS
LIN {X -0.017,Y -321.918,Z 1332.690,A 0.000,B 0.000,C 90.000,E1 124.119} C_DIS
LIN {X -0.066,Y -323.457,Z 1332.688,A 0.000,B 0.000,C 90.000,E1 123.833} C_DIS
LIN {X 0.109,Y -325.867,Z 1332.684,A 0.000,B 0.000,C 90.000,E1 123.166} C_DIS
LIN {X 0.112,Y -336.340,Z 1332.669,A 0.000,B 0.000,C 90.000,E1 120.335} C_DIS
LIN {X -0.098,Y -348.162,Z 1332.653,A 0.000,B 0.000,C 90.000,E1 117.590} C_DIS
LIN {X 0.025,Y -361.427,Z 1332.638,A 0.000,B 0.000,C 90.000,E1 114.847} C_DIS
LIN {X 0.128,Y -374.529,Z 1332.625,A 0.000,B 0.000,C 90.000,E1 112.461} C_DIS
LIN {X -0.091,Y -388.957,Z 1332.612,A 0.000,B 0.000,C 90.000,E1 110.174} C_DIS
LIN {X 0.142,Y -404.812,Z 1332.599,A 0.000,B 0.000,C 90.000,E1 107.873} C_DIS
LIN {X 0.146,Y -422.205,Z 1332.587,A 0.000,B 0.000,C 90.000,E1 105.662} C_DIS
LIN {X -0.041,Y -441.236,Z 1332.575,A 0.000,B 0.000,C 90.000,E1 103.536} C_DIS
LIN {X -0.180,Y -461.287,Z 1332.564,A 0.000,B 0.000,C 90.000,E1 101.535} C_DIS
LIN {X -0.205,Y -479.268,Z 1332.555,A 0.000,B 0.000,C 90.000,E1 99.905} C_DIS
LIN {X -0.131,Y -481.358,Z 1332.554,A 0.000,B 0.000,C 90.000,E1 99.670} C_DIS
LIN {X -0.136,Y -482.947,Z 1332.552,A 0.000,B 0.000,C 90.000,E1 99.443} C_DIS
LIN {X -0.253,Y -484.277,Z 1332.551,A 0.000,B 0.000,C 90.000,E1 99.208} C_DIS
LIN {X 0.108,Y -485.258,Z 1332.550,A 0.000,B 0.000,C 90.000,E1 98.916} C_DIS
LIN {X -0.187,Y -486.356,Z 1332.547,A 0.000,B 0.000,C 90.000,E1 98.454} C_DIS
LIN {X 0.007,Y -486.447,Z 1332.544,A 0.000,B 0.000,C 90.000,E1 97.936} C_DIS
LIN {X -0.211,Y -485.548,Z 1332.541,A 0.000,B 0.000,C 90.000,E1 97.466} C_DIS
LIN {X -0.011,Y -483.506,Z 1332.539,A 0.000,B 0.000,C 90.000,E1 96.947} C_DIS
LIN {X -0.183,Y -481.923,Z 1332.537,A 0.000,B 0.000,C 90.000,E1 96.720} C_DIS
LIN {X -0.168,Y -471.014,Z 1332.529,A 0.000,B 0.000,C 90.000,E1 95.220} C_DIS
LIN {X 0.107,Y -457.476,Z 1332.518,A 0.000,B 0.000,C 90.000,E1 93.154} C_DIS
LIN {X -0.184,Y -442.601,Z 1332.505,A 0.000,B 0.000,C 90.000,E1 90.859} C_DIS
LIN {X -0.132,Y -426.126,Z 1332.488,A 0.000,B 0.000,C 90.000,E1 87.936} C_DIS
LIN {X -0.136,Y -416.070,Z 1332.478,A 0.000,B 0.000,C 90.000,E1 86.045} C_DIS
LIN {X 0.104,Y -405.778,Z 1332.467,A 0.000,B 0.000,C 90.000,E1 84.090} C_DIS
LIN {X 0.147,Y -396.822,Z 1332.458,A 0.000,B 0.000,C 90.000,E1 82.413} C_DIS
LIN {X 0.032,Y -387.591,Z 1332.449,A 0.000,B 0.000,C 90.000,E1 80.735} C_DIS
LIN {X -0.183,Y -378.156,Z 1332.439,A 0.000,B 0.000,C 90.000,E1 79.050} C_DIS
LIN {X -0.050,Y -366.865,Z 1332.428,A 0.000,B 0.000,C 90.000,E1 76.992} C_DIS
LIN {X -0.164,Y -355.360,Z 1332.416,A 0.000,B 0.000,C 90.000,E1 74.936} C_DIS
LIN {X 0.097,Y -343.814,Z 1332.404,A 0.000,B 0.000,C 90.000,E1 72.779} C_DIS
LIN {X 0.204,Y -332.182,Z 1332.392,A 0.000,B 0.000,C 90.000,E1 70.604} C_DIS
LIN {X 0.118,Y -319.193,Z 1332.378,A 0.000,B 0.000,C 90.000,E1 68.103} C_DIS
LIN {X -0.081,Y -302.504,Z 1332.359,A 0.000,B 0.000,C 90.000,E1 64.588} C_DIS
LIN {X -0.119,Y -293.027,Z 1332.346,A 0.000,B 0.000,C 90.000,E1 62.281} C_DIS
LIN {X -0.059,Y -285.796,Z 1332.335,A 0.000,B 0.000,C 90.000,E1 60.255} C_DIS
LIN {X -0.063,Y -274.266,Z 1332.314,A 0.000,B 0.000,C 90.000,E1 56.501} C_DIS
LIN {X 0.004,Y -264.899,Z 1332.294,A 0.000,B 0.000,C 90.000,E1 53.004} C_DIS
LIN {X -0.003,Y -256.084,Z 1332.275,A 0.000,B 0.000,C 90.000,E1 49.461} C_DIS
LIN {X -0.160,Y -247.809,Z 1332.255,A 0.000,B 0.000,C 90.000,E1 45.891} C_DIS
LIN {X -0.061,Y -239.965,Z 1332.234,A 0.000,B 0.000,C 90.000,E1 42.204} C_DIS
LIN {X 0.020,Y -232.807,Z 1332.214,A 0.000,B 0.000,C 90.000,E1 38.463} C_DIS
LIN {X 0.004,Y -226.552,Z 1332.193,A 0.000,B 0.000,C 90.000,E1 34.692} C_DIS
LIN {X -0.022,Y -221.300,Z 1332.172,A 0.000,B 0.000,C 90.000,E1 30.875} C_DIS
LIN {X -0.011,Y -216.342,Z 1332.146,A 0.000,B 0.000,C 90.000,E1 26.232} C_DIS
LIN {X 0.023,Y -212.349,Z 1332.120,A 0.000,B 0.000,C 90.000,E1 21.535} C_DIS
LIN {X 0.084,Y -209.441,Z 1332.098,A 0.000,B 0.000,C 90.000,E1 17.583} C_DIS
LIN {X 0.053,Y -207.295,Z 1332.080,A 0.000,B 0.000,C 90.000,E1 14.426} C_DIS
LIN {X 0.061,Y -205.250,Z 1332.063,A 0.000,B 0.000,C 90.000,E1 11.243} C_DIS
LIN {X -0.076,Y -202.306,Z 1332.031,A 0.000,B 0.000,C 90.000,E1 5.682} C_DIS
LIN {X -0.052,Y -200.254,Z 1331.993,A 0.000,B 0.000,C 90.000,E1 358.740} C_DIS
LIN {X 0.084,Y -200.260,Z 1331.957,A 0.000,B 0.000,C 90.000,E1 352.243} C_DIS
LIN {X -0.027,Y -202.227,Z 1331.921,A 0.000,B 0.000,C 90.000,E1 345.825} C_DIS
LIN {X 0.053,Y -205.697,Z 1331.890,A 0.000,B 0.000,C 90.000,E1 340.188} C_DIS
LIN {X -0.029,Y -209.315,Z 1331.868,A 0.000,B 0.000,C 90.000,E1 336.230} C_DIS
LIN {X -0.033,Y -213.898,Z 1331.846,A 0.000,B 0.000,C 90.000,E1 332.281} C_DIS
LIN {X 0.136,Y -219.502,Z 1331.824,A 0.000,B 0.000,C 90.000,E1 328.329} C_DIS
LIN {X 0.083,Y -226.156,Z 1331.803,A 0.000,B 0.000,C 90.000,E1 324.482} C_DIS
LIN {X -0.011,Y -232.229,Z 1331.786,A 0.000,B 0.000,C 90.000,E1 321.457} C_DIS
LIN {X -0.075,Y -240.882,Z 1331.765,A 0.000,B 0.000,C 90.000,E1 317.715} C_DIS
LIN {X 0.097,Y -249.636,Z 1331.747,A 0.000,B 0.000,C 90.000,E1 314.352} C_DIS
LIN {X 0.015,Y -258.666,Z 1331.730,A 0.000,B 0.000,C 90.000,E1 311.472} C_DIS
LIN {X -0.047,Y -267.601,Z 1331.717,A 0.000,B 0.000,C 90.000,E1 308.991} C_DIS
LIN {X 0.069,Y -279.308,Z 1331.701,A 0.000,B 0.000,C 90.000,E1 306.171} C_DIS
LIN {X 0.050,Y -289.212,Z 1331.690,A 0.000,B 0.000,C 90.000,E1 304.119} C_DIS
LIN {X 0.138,Y -298.345,Z 1331.680,A 0.000,B 0.000,C 90.000,E1 302.418} C_DIS
LIN {X -0.046,Y -308.460,Z 1331.671,A 0.000,B 0.000,C 90.000,E1 300.797} C_DIS
LIN {X -0.024,Y -317.401,Z 1331.664,A 0.000,B 0.000,C 90.000,E1 299.489} C_DIS
LIN {X -0.067,Y -329.547,Z 1331.655,A 0.000,B 0.000,C 90.000,E1 297.897} C_DIS
LIN {X 0.074,Y -347.750,Z 1331.643,A 0.000,B 0.000,C 90.000,E1 295.720} C_DIS
LIN {X -0.004,Y -360.728,Z 1331.635,A 0.000,B 0.000,C 90.000,E1 294.259} C_DIS
LIN {X 0.011,Y -371.165,Z 1331.628,A 0.000,B 0.000,C 90.000,E1 293.078} C_DIS
LIN {X 0.225,Y -383.734,Z 1331.620,A 0.000,B 0.000,C 90.000,E1 291.589} C_DIS
LIN {X 0.132,Y -398.379,Z 1331.611,A 0.000,B 0.000,C 90.000,E1 289.885} C_DIS
LIN {X 0.047,Y -415.569,Z 1331.600,A 0.000,B 0.000,C 90.000,E1 287.946} C_DIS
LIN {X 0.006,Y -425.167,Z 1331.594,A 0.000,B 0.000,C 90.000,E1 286.858} C_DIS
LIN {X -0.064,Y -434.118,Z 1331.588,A 0.000,B 0.000,C 90.000,E1 285.788} C_DIS
LIN {X 0.193,Y -440.219,Z 1331.583,A 0.000,B 0.000,C 90.000,E1 284.954} C_DIS
LIN {X 0.083,Y -445.674,Z 1331.579,A 0.000,B 0.000,C 90.000,E1 284.175} C_DIS
LIN {X -0.098,Y -450.407,Z 1331.574,A 0.000,B 0.000,C 90.000,E1 283.411} C_DIS
LIN {X 0.209,Y -454.444,Z 1331.570,A 0.000,B 0.000,C 90.000,E1 282.591} C_DIS
LIN {X 0.107,Y -457.689,Z 1331.566,A 0.000,B 0.000,C 90.000,E1 281.827} C_DIS
LIN {X 0.205,Y -459.388,Z 1331.563,A 0.000,B 0.000,C 90.000,E1 281.299} C_DIS
LIN {X -0.231,Y -460.762,Z 1331.560,A 0.000,B 0.000,C 90.000,E1 280.838} C_DIS
LIN {X -0.118,Y -461.746,Z 1331.557,A 0.000,B 0.000,C 90.000,E1 280.310} C_DIS
LIN {X -0.079,Y -462.354,Z 1331.554,A 0.000,B 0.000,C 90.000,E1 279.792} C_DIS
LIN {X 0.046,Y -462.514,Z 1331.552,A 0.000,B 0.000,C 90.000,E1 279.265} C_DIS
LIN {X 0.100,Y -462.203,Z 1331.549,A 0.000,B 0.000,C 90.000,E1 278.746} C_DIS
LIN {X 0.223,Y -461.516,Z 1331.546,A 0.000,B 0.000,C 90.000,E1 278.219} C_DIS
LIN {X -0.181,Y -460.264,Z 1331.543,A 0.000,B 0.000,C 90.000,E1 277.757} C_DIS
LIN {X -0.129,Y -458.491,Z 1331.540,A 0.000,B 0.000,C 90.000,E1 277.239} C_DIS
LIN {X -0.084,Y -456.197,Z 1331.537,A 0.000,B 0.000,C 90.000,E1 276.720} C_DIS
LIN {X -0.054,Y -453.338,Z 1331.534,A 0.000,B 0.000,C 90.000,E1 276.201} C_DIS
LIN {X -0.041,Y -449.889,Z 1331.531,A 0.000,B 0.000,C 90.000,E1 275.682} C_DIS
LIN {X -0.046,Y -445.734,Z 1331.529,A 0.000,B 0.000,C 90.000,E1 275.163} C_DIS
LIN {X -0.074,Y -440.660,Z 1331.526,A 0.000,B 0.000,C 90.000,E1 274.645} C_DIS
LIN {X 0.029,Y -434.807,Z 1331.523,A 0.000,B 0.000,C 90.000,E1 274.131} C_DIS
LIN {X 0.165,Y -428.765,Z 1331.521,A 0.000,B 0.000,C 90.000,E1 273.669} C_DIS
LIN {X 0.189,Y -422.251,Z 1331.518,A 0.000,B 0.000,C 90.000,E1 273.269} C_DIS
LIN {X 0.199,Y -415.703,Z 1331.516,A 0.000,B 0.000,C 90.000,E1 272.922} C_DIS
LIN {X 0.079,Y -409.118,Z 1331.515,A 0.000,B 0.000,C 90.000,E1 272.636} C_DIS
LIN {X 0.185,Y -402.195,Z 1331.513,A 0.000,B 0.000,C 90.000,E1 272.350} C_DIS
LIN {X 0.152,Y -394.698,Z 1331.512,A 0.000,B 0.000,C 90.000,E1 272.121} C_DIS
LIN {X 0.051,Y -387.110,Z 1331.511,A 0.000,B 0.000,C 90.000,E1 271.949} C_DIS
LIN {X -0.175,Y -379.501,Z 1331.510,A 0.000,B 0.000,C 90.000,E1 271.833} C_DIS
LIN {X 0.137,Y -371.014,Z 1331.509,A 0.000,B 0.000,C 90.000,E1 271.661} C_DIS
LIN {X 0.130,Y -357.521,Z 1331.509,A 0.000,B 0.000,C 90.000,E1 271.547} C_DIS
LIN {X -0.045,Y -349.743,Z 1331.509,A 0.000,B 0.000,C 90.000,E1 271.547} C_DIS
LIN {X -0.053,Y -181.346,Z 1331.509,A 0.000,B 0.000,C 90.000,E1 271.547} C_DIS
LIN {X -0.006,Y -181.560,Z 1331.500,A 0.000,B 0.000,C 90.000,E1 270.000} C_DIS
LIN {X -0.051,Y -180.903,Z 1331.474,A 0.000,B 0.000,C 90.000,E1 265.298} C_DIS
LIN {X 0.079,Y -180.236,Z 1331.464,A 0.000,B 0.000,C 90.000,E1 263.571} C_DIS
LIN {X -0.081,Y -178.721,Z 1331.441,A 0.000,B 0.000,C 90.000,E1 259.398} C_DIS
LIN {X -0.013,Y -175.770,Z 1331.413,A 0.000,B 0.000,C 90.000,E1 254.283} C_DIS
LIN {X 0.036,Y -171.953,Z 1331.384,A 0.000,B 0.000,C 90.000,E1 249.135} C_DIS
LIN {X 0.013,Y -171.343,Z 1331.379,A 0.000,B 0.000,C 90.000,E1 248.284} C_DIS
LIN {X -0.009,Y -167.596,Z 1331.355,A 0.000,B 0.000,C 90.000,E1 243.973} C_DIS
LIN {X 0.003,Y -166.237,Z 1331.346,A 0.000,B 0.000,C 90.000,E1 242.231} C_DIS
LIN {X -0.008,Y -162.995,Z 1331.326,A 0.000,B 0.000,C 90.000,E1 238.742} C_DIS
LIN {X 0.038,Y -160.915,Z 1331.312,A 0.000,B 0.000,C 90.000,E1 236.087} C_DIS
LIN {X 0.016,Y -157.678,Z 1331.292,A 0.000,B 0.000,C 90.000,E1 232.557} C_DIS
LIN {X -0.046,Y -155.717,Z 1331.277,A 0.000,B 0.000,C 90.000,E1 229.908} C_DIS
LIN {X 0.009,Y -151.978,Z 1331.252,A 0.000,B 0.000,C 90.000,E1 225.405} C_DIS
LIN {X 0.025,Y -150.221,Z 1331.237,A 0.000,B 0.000,C 90.000,E1 222.690} C_DIS
LIN {X -0.051,Y -146.985,Z 1331.212,A 0.000,B 0.000,C 90.000,E1 218.177} C_DIS
LIN {X 0.057,Y -145.571,Z 1331.197,A 0.000,B 0.000,C 90.000,E1 215.391} C_DIS
LIN {X 0.056,Y -142.961,Z 1331.171,A 0.000,B 0.000,C 90.000,E1 210.797} C_DIS
LIN {X -0.013,Y -141.587,Z 1331.151,A 0.000,B 0.000,C 90.000,E1 207.129} C_DIS
LIN {X 0.034,Y -139.419,Z 1331.115,A 0.000,B 0.000,C 90.000,E1 200.610} C_DIS
LIN {X -0.046,Y -139.144,Z 1331.104,A 0.000,B 0.000,C 90.000,E1 198.779} C_DIS
LIN {X -0.024,Y -138.347,Z 1331.057,A 0.000,B 0.000,C 90.000,E1 190.366} C_DIS
LIN {X -0.038,Y -139.490,Z 1331.006,A 0.000,B 0.000,C 90.000,E1 181.031} C_DIS
LIN {X 0.043,Y -141.097,Z 1330.975,A 0.000,B 0.000,C 90.000,E1 175.412} C_DIS
LIN {X -0.004,Y -142.474,Z 1330.959,A 0.000,B 0.000,C 90.000,E1 172.648} C_DIS
LIN {X -0.057,Y -144.721,Z 1330.933,A 0.000,B 0.000,C 90.000,E1 168.049} C_DIS
LIN {X 0.036,Y -147.323,Z 1330.913,A 0.000,B 0.000,C 90.000,E1 164.338} C_DIS
LIN {X -0.039,Y -150.646,Z 1330.888,A 0.000,B 0.000,C 90.000,E1 159.806} C_DIS
LIN {X -0.016,Y -154.123,Z 1330.868,A 0.000,B 0.000,C 90.000,E1 156.177} C_DIS
LIN {X -0.093,Y -157.549,Z 1330.848,A 0.000,B 0.000,C 90.000,E1 152.615} C_DIS
LIN {X 0.072,Y -161.789,Z 1330.828,A 0.000,B 0.000,C 90.000,E1 148.997} C_DIS
LIN {X -0.045,Y -165.982,Z 1330.808,A 0.000,B 0.000,C 90.000,E1 145.515} C_DIS
LIN {X -0.049,Y -170.978,Z 1330.789,A 0.000,B 0.000,C 90.000,E1 142.029} C_DIS
LIN {X 0.002,Y -175.847,Z 1330.770,A 0.000,B 0.000,C 90.000,E1 138.566} C_DIS
LIN {X -0.004,Y -181.451,Z 1330.751,A 0.000,B 0.000,C 90.000,E1 135.162} C_DIS
LIN {X -0.131,Y -186.961,Z 1330.732,A 0.000,B 0.000,C 90.000,E1 131.838} C_DIS
LIN {X -0.010,Y -190.075,Z 1330.723,A 0.000,B 0.000,C 90.000,E1 130.135} C_DIS
